// TwinCAT 3 PLC project TCP
// Title: Tc_TcpIpDevices
// Company: NewEngineer
// Author: https://github.com/phucpha
// ProjectVersion: 0.0.0.1
// Description: TC_TcpIpDevices use for Device that communicate by TCPIP.
// ProgramVersion: 3.1.4024.0
// libraries:
//   Tc2_Standard, * (Beckhoff Automation GmbH)
//   Tc2_System, * (Beckhoff Automation GmbH)
//   Tc2_TcpIp, * (Beckhoff Automation GmbH)
//   Tc3_EventLogger, * (Beckhoff Automation GmbH)
//   Tc3_Module, * (Beckhoff Automation GmbH)
//   Tc_Utilities, * (NewEngineer)
// project tree:
//   DUTs/Cognex/ E_CognexCameraGetConnectionStatus.TcDUT, E_CognexCameraGetExprStatus.TcDUT, E_CognexCameraGetFileListStatus.TcDUT, E_CognexCameraGetFileStatus.TcDUT, E_CognexCameraGetJobStatus.TcDUT, E_CognexCameraGetOnlineStatus.TcDUT, E_CognexCameraGetPositionState.TcDUT, E_CognexCameraGetPositionStatus.TcDUT, E_CognexCameraGetValueEasyBuilderStatus.TcDUT, E_CognexCameraGetValueSpreadsheetStatus.TcDUT, E_CognexCameraGetValuesState.TcDUT, E_CognexCameraGetValuesStatus.TcDUT, E_CognexCameraGetValueStatus.TcDUT, E_CognexCameraImageTriggerStatus.TcDUT, E_CognexCameraInitState.TcDUT, E_CognexCameraLoadFileStatus.TcDUT, E_CognexCameraMethodState.TcDUT, E_CognexCameraPutLiveStatus.TcDUT, E_CognexCameraPutPortnumStatus.TcDUT, E_CognexCameraPutTimeoutStatus.TcDUT, E_CognexCameraPutUpdateStatus.TcDUT, E_CognexCameraPutWatchStatus.TcDUT, E_CognexCameraResetSystemStatus.TcDUT, E_CognexCameraSetJobStatus.TcDUT, E_CognexCameraSetOnlineStatus.TcDUT, E_CognexCameraState.TcDUT, E_CognexCameraStoreFileStatus.TcDUT
//   DUTs/TcpIp/ E_TcpIpDeviceState.TcDUT, E_TcpIpDeviceStateRecive.TcDUT, E_TcpIpDeviceStateSend.TcDUT, E_TcpIpServerStateRunning.TcDUT, ST_TcpBufferData.TcDUT
//   FC/ FUN_StringToTcpBufferData.TcPOU, FUN_TcpBufferDataToString.TcPOU
//   / PlcTask.TcTTO
//   POUs/Base/Tcp Buffer/ FB_TcpBuffer.TcPOU
//   POUs/Base/Tcp Client/ FB_TcpClient.TcPOU
//   POUs/Base/Tcp Device/ FB_TcpDevice.TcPOU, I_TcpDevice.TcIO
//   POUs/Base/Tcp Server/ FB_TcpServer.TcPOU
//   POUs/Cognex/ FB_CognexCamera.TcPOU, I_CognexCamera.TcIO
//   Version/ Global_Version.TcGVL
// real-time tasks:
//   TASK PlcTask: cycle T#10ms, priority 20, ADS port 350

CONFIGURATION TCP
    RESOURCE PLC ON TwinCAT3
        TASK PlcTask(INTERVAL := T#10ms, PRIORITY := 20);
    END_RESOURCE
END_CONFIGURATION

// ---- DUTs/Cognex/E_CognexCameraGetConnectionStatus.TcDUT
{attribute 'strict'}
TYPE E_CognexCameraGetConnectionStatus :
(
	WAITING_FOR_STATUS_CODE						:= 2,
	THE_COMMAND_WAS_EXECUTED_SUCCESSFULLY		:= 1,
	UNRECOGNIZED_COMMAND 						:= 0,
	THE_CELL_ID_IS_INVALID						:= -1,
	THE_COMMAND_COULD_NOT_BE_EXECUTED 			:= -2,
	USER_DOES_NOT_HAVE_FULL_ACCESS				:= -6
);
END_TYPE

// ---- DUTs/Cognex/E_CognexCameraGetExprStatus.TcDUT
{attribute 'strict'}
TYPE E_CognexCameraGetExprStatus :
(
	WAITING_FOR_STATUS_CODE										:= 2,
	THE_COMMAND_WAS_EXECUTED_SUCCESSFULLY						:= 1,
	UNRECOGNIZED_COMMAND 										:= 0,
	THE_CELL_ID_IS_INVALID_OR_HAS_EXCEEDED_15_BYTES_IN_LENGTH	:= -1,
	THE_COMMAND_COULD_NOT_BE_EXECUTED 							:= -2
);
END_TYPE

// ---- DUTs/Cognex/E_CognexCameraGetFileListStatus.TcDUT
{attribute 'strict'}
TYPE E_CognexCameraGetFileListStatus :
(
	WAITING_FOR_STATUS_CODE									:= 2,
	THE_COMMAND_WAS_EXECUTED_SUCCESSFULLY					:= 1,
	UNRECOGNIZED_COMMAND 									:= 0,
	THE_INPUT_IS_INVALID_OR_HAS_EXCEEDED_15_BYTES_IN_LENGTH	:= -1,
	THE_ACTIVE_JOB_HAS_NOT_BEEN_SAVED 						:= -2
);
END_TYPE

// ---- DUTs/Cognex/E_CognexCameraGetFileStatus.TcDUT
{attribute 'strict'}
TYPE E_CognexCameraGetFileStatus :
(
	WAITING_FOR_STATUS_CODE						:= 2,
	THE_COMMAND_WAS_EXECUTED_SUCCESSFULLY		:= 1,
	UNRECOGNIZED_COMMAND 						:= 0,
	THE_ACTIVE_JOB_HAS_NOT_BEEN_SAVED 			:= -2
);
END_TYPE

// ---- DUTs/Cognex/E_CognexCameraGetJobStatus.TcDUT
{attribute 'strict'}
TYPE E_CognexCameraGetJobStatus :
(
	WAITING_FOR_STATUS_CODE														:= 2,
	THE_COMMAND_WAS_EXECUTED_SUCCESSFULLY										:= 1,
	UNRECOGNIZED_COMMAND 														:= 0,
	THE_ACTIVE_JOB_HAS_NOT_BEEN_SAVED_OR_DOES_NOT_HAVE_A_NUMERICAL_PREFIX		:= -2
);
END_TYPE

// ---- DUTs/Cognex/E_CognexCameraGetOnlineStatus.TcDUT
{attribute 'strict'}
TYPE E_CognexCameraGetOnlineStatus :
(
	WAITING_FOR_STATUS_CODE								:= 2,
	THE_IN_SIGHT_VISION_SYSTEM_IS_CURRENTLY_OFFLINE		:= 0,
	THE_IN_SIGHT_VISION_SYSTEM_IS_CURRENTLY_ONLINE 		:= 1
);
END_TYPE

// ---- DUTs/Cognex/E_CognexCameraGetPositionState.TcDUT
{attribute 'strict'}
TYPE E_CognexCameraGetPositionState :
(
	CAMERA_GET_POSITION_SEND_COMMAND_X				:= 0,
	CAMERA_GET_POSITION_RECEIVE_RESPONSE_X			:= 10,
	CAMERA_GET_POSITION_SEND_COMMAND_Y				:= 20,
	CAMERA_GET_POSITION_RECEIVE_RESPONSE_Y			:= 30,
	CAMERA_GET_POSITION_SEND_COMMAND_ROTATION		:= 40,
	CAMERA_GET_POSITION_RECEIVE_RESPONSE_ROTATION	:= 50,
	CAMERA_GET_POSITION_GETTING_DONE				:= 60
);
END_TYPE

// ---- DUTs/Cognex/E_CognexCameraGetPositionStatus.TcDUT
{attribute 'strict'}
TYPE E_CognexCameraGetPositionStatus :
(
	WAITING_FOR_STATUS_CODE						:= 2,
	THE_COMMAND_WAS_EXECUTED_SUCCESSFULLY		:= 1,
	UNRECOGNIZED_COMMAND 						:= 0,
	THE_SYMBOLIC_TAG_IS_INVALID					:= -1,
	THE_COMMAND_COULD_NOT_BE_EXECUTED 			:= -2,
	PRODUCT_NOT_FOUND							:= -3
);
END_TYPE

// ---- DUTs/Cognex/E_CognexCameraGetValueEasyBuilderStatus.TcDUT
{attribute 'strict'}
TYPE E_CognexCameraGetValueEasyBuilderStatus :
(
	WAITING_FOR_STATUS_CODE						:= 2,
	THE_COMMAND_WAS_EXECUTED_SUCCESSFULLY		:= 1,
	UNRECOGNIZED_COMMAND 						:= 0,
	THE_SYMBOLIC_TAG_IS_INVALID					:= -1,
	THE_COMMAND_COULD_NOT_BE_EXECUTED 			:= -2
);
END_TYPE

// ---- DUTs/Cognex/E_CognexCameraGetValueSpreadsheetStatus.TcDUT
{attribute 'strict'}
TYPE E_CognexCameraGetValueSpreadsheetStatus :
(
	WAITING_FOR_STATUS_CODE						:= 2,
	THE_COMMAND_WAS_EXECUTED_SUCCESSFULLY		:= 1,
	UNRECOGNIZED_COMMAND 						:= 0,
	THE_CELL_ID_IS_INVALID						:= -1,
	THE_COMMAND_COULD_NOT_BE_EXECUTED 			:= -2
);
END_TYPE

// ---- DUTs/Cognex/E_CognexCameraGetValuesState.TcDUT
{attribute 'strict'}
TYPE E_CognexCameraGetValuesState :
(
	CAMERA_GET_VALUES_SEND_COMMAND_VALUE_1		:= 0,
	CAMERA_GET_VALUES_RECEIVE_RESPONSE_VALUE_1	:= 10,
	CAMERA_GET_VALUES_SEND_COMMAND_VALUE_2		:= 20,
	CAMERA_GET_VALUES_RECEIVE_RESPONSE_VALUE_2	:= 30,
	CAMERA_GET_VALUES_SEND_COMMAND_VALUE_3		:= 40,
	CAMERA_GET_VALUES_RECEIVE_RESPONSE_VALUE_3	:= 50,
	CAMERA_GET_VALUES_SEND_COMMAND_VALUE_4		:= 60,
	CAMERA_GET_VALUES_RECEIVE_RESPONSE_VALUE_4	:= 70,
	CAMERA_GET_VALUES_GETTING_DONE				:= 80
);
END_TYPE

// ---- DUTs/Cognex/E_CognexCameraGetValuesStatus.TcDUT
{attribute 'strict'}
TYPE E_CognexCameraGetValuesStatus :
(
	WAITING_FOR_STATUS_CODE						:= 2,
	THE_COMMAND_WAS_EXECUTED_SUCCESSFULLY		:= 1,
	UNRECOGNIZED_COMMAND 						:= 0,
	THE_SYMBOLIC_TAG_IS_INVALID					:= -1,
	THE_COMMAND_COULD_NOT_BE_EXECUTED 			:= -2,
	ONE_OR_MORE_VALUE_IS_INVALID				:= -3
);
END_TYPE

// ---- DUTs/Cognex/E_CognexCameraGetValueStatus.TcDUT
{attribute 'strict'}
TYPE E_CognexCameraGetValueStatus :
(
	WAITING_FOR_STATUS_CODE						:= 2,
	THE_COMMAND_WAS_EXECUTED_SUCCESSFULLY		:= 1,
	UNRECOGNIZED_COMMAND 						:= 0,
	THE_CELL_ID_IS_INVALID						:= -1,
	THE_COMMAND_COULD_NOT_BE_EXECUTED 			:= -2,
	USER_DOES_NOT_HAVE_FULL_ACCESS				:= -6
);
END_TYPE

// ---- DUTs/Cognex/E_CognexCameraImageTriggerStatus.TcDUT
{attribute 'strict'}
TYPE E_CognexCameraImageTriggerStatus :
(
	WAITING_FOR_STATUS_CODE										:= 2,
	THE_COMMAND_WAS_EXECUTED_SUCCESSFULLY						:= 1,
	UNRECOGNIZED_COMMAND 										:= 0,
	THE_NUMBER_IS_EITHER_OUT_OF_RANGE_OR_NOT_AN_INTEGER 		:= -1,
	THE_COMMAND_COULD_NOT_BE_EXECUTED_OR_THE_SENSOR_IS_OFFLINE 	:= -2,
	USER_DOES_NOT_HAVE_FULL_ACCESS								:= -6
);
END_TYPE

// ---- DUTs/Cognex/E_CognexCameraInitState.TcDUT
{attribute 'strict'}
TYPE E_CognexCameraInitState :
(
	CAMERA_INIT_CONNECTION 				:= 0,
	CAMERA_INIT_CLEAR_BUFFER			:= 10,	
	CAMERA_INIT_WAIT_FOR_USERNAME 		:= 20,	
	CAMERA_INIT_WRITE_USER				:= 30,	
	CAMERA_INIT_WAIT_FOR_PASSWORD 		:= 40,	
	CAMERA_INIT_WRITE_PASSWORD			:= 50,	
	CAMERA_INIT_WAIT_FOR_CONFIRMATION	:= 60,
	CAMERA_INIT_DONE					:= 80
);
END_TYPE

// ---- DUTs/Cognex/E_CognexCameraLoadFileStatus.TcDUT
{attribute 'strict'}
TYPE E_CognexCameraLoadFileStatus :
(
	WAITING_FOR_STATUS_CODE						:= 2,
	THE_COMMAND_WAS_EXECUTED_SUCCESSFULLY		:= 1,
	UNRECOGNIZED_COMMAND 						:= 0,
	THE_FILENAME_IS_MISSING						:= -1,
	THE_JOB_FAILED_TO_LOAD 						:= -2,
	THE_VISION_SYSTEM_IS_OUT_OF_MEMORY			:= -4,
	USER_DOES_NOT_HAVE_FULL_ACCESS				:= -6
);
END_TYPE

// ---- DUTs/Cognex/E_CognexCameraMethodState.TcDUT
{attribute 'strict'}
TYPE E_CognexCameraMethodState :
(
	CAMERA_METHOD_SEND_COMMAND 			:= 0,
	CAMERA_METHOD_RECEIVE_RESPONSE 		:= 10
);
END_TYPE

// ---- DUTs/Cognex/E_CognexCameraPutLiveStatus.TcDUT
{attribute 'strict'}
TYPE E_CognexCameraPutLiveStatus :
(
	WAITING_FOR_STATUS_CODE										:= 2,
	THE_COMMAND_WAS_EXECUTED_SUCCESSFULLY						:= 1,
	UNRECOGNIZED_COMMAND 										:= 0,
	THE_INPUT_IS_INVALID_OR_HAS_EXCEEDED_15_BYTES_IN_LENGTH		:= -1,
	THE_COMMAND_COULD_NOT_BE_EXECUTED 							:= -2,
	USER_DOES_NOT_HAVE_FULL_ACCESS	 							:= -6
);
END_TYPE

// ---- DUTs/Cognex/E_CognexCameraPutPortnumStatus.TcDUT
{attribute 'strict'}
TYPE E_CognexCameraPutPortnumStatus :
(
	WAITING_FOR_STATUS_CODE										:= 2,
	THE_COMMAND_WAS_EXECUTED_SUCCESSFULLY						:= 1,
	UNRECOGNIZED_COMMAND 										:= 0,
	THE_INPUT_IS_INVALID_OR_HAS_EXCEEDED_15_BYTES_IN_LENGTH		:= -1,
	THE_COMMAND_COULD_NOT_BE_EXECUTED 							:= -2,
	USER_DOES_NOT_HAVE_FULL_ACCESS	 							:= -6
);
END_TYPE

// ---- DUTs/Cognex/E_CognexCameraPutTimeoutStatus.TcDUT
{attribute 'strict'}
TYPE E_CognexCameraPutTimeoutStatus :
(
	WAITING_FOR_STATUS_CODE										:= 2,	
	THE_COMMAND_WAS_EXECUTED_SUCCESSFULLY						:= 1,
	UNRECOGNIZED_COMMAND 										:= 0,
	THE_INPUT_IS_INVALID_OR_HAS_EXCEEDED_15_BYTES_IN_LENGTH		:= -1,
	USER_DOES_NOT_HAVE_FULL_ACCESS	 							:= -6
);
END_TYPE

// ---- DUTs/Cognex/E_CognexCameraPutUpdateStatus.TcDUT
{attribute 'strict'}
TYPE E_CognexCameraPutUpdateStatus :
(
	WAITING_FOR_STATUS_CODE										:= 2,	
	THE_COMMAND_WAS_EXECUTED_SUCCESSFULLY						:= 1,
	UNRECOGNIZED_COMMAND 										:= 0,
	THE_INPUT_IS_INVALID_OR_HAS_EXCEEDED_15_BYTES_IN_LENGTH		:= -1,
	THE_COMMAND_COULD_NOT_BE_EXECUTED 							:= -2,
	USER_DOES_NOT_HAVE_FULL_ACCESS	 							:= -6
);
END_TYPE

// ---- DUTs/Cognex/E_CognexCameraPutWatchStatus.TcDUT
{attribute 'strict'}
TYPE E_CognexCameraPutWatchStatus :
(
	WAITING_FOR_STATUS_CODE										:= 2,	
	THE_COMMAND_WAS_EXECUTED_SUCCESSFULLY						:= 1,
	UNRECOGNIZED_COMMAND 										:= 0,
	THE_INPUT_IS_INVALID_OR_HAS_EXCEEDED_15_BYTES_IN_LENGTH		:= -1,
	THE_COMMAND_COULD_NOT_BE_EXECUTED 							:= -2,
	USER_DOES_NOT_HAVE_FULL_ACCESS								:= -6
);
END_TYPE

// ---- DUTs/Cognex/E_CognexCameraResetSystemStatus.TcDUT
{attribute 'strict'}
TYPE E_CognexCameraResetSystemStatus :
(
	WAITING_FOR_STATUS_CODE					:= 2,	
	THE_COMMAND_WAS_EXECUTED_SUCCESSFULLY	:= -1,
	USER_DOES_NOT_HAVE_FULL_ACCESS			:= -6
);
END_TYPE

// ---- DUTs/Cognex/E_CognexCameraSetJobStatus.TcDUT
{attribute 'strict'}
TYPE E_CognexCameraSetJobStatus :
(
	WAITING_FOR_STATUS_CODE														:= 2,	
	THE_COMMAND_WAS_EXECUTED_SUCCESSFULLY										:= 1,
	UNRECOGNIZED_COMMAND 														:= 0,
	THE_ID_IS_LESS_THAN_0_OR_IS_NOT_AN_INTEGER									:= -1,
	THE_JOB_FAILED_TO_LOAD_THE_SENSOR_IS_ONLINE_OR_THE_FILE_WAS_NOT_FOUND		:= -2,
	THE_IN_SIGHT_SENSOR_IS_OUT_OF_MEMORY										:= -4,
	USER_DOES_NOT_HAVE_FULL_ACCESS												:= -6
);
END_TYPE

// ---- DUTs/Cognex/E_CognexCameraSetOnlineStatus.TcDUT
{attribute 'strict'}
TYPE E_CognexCameraSetOnlineStatus :
(
	WAITING_FOR_STATUS_CODE																		:= 2,	
	THE_COMMAND_WAS_EXECUTED_SUCCESSFULLY														:= 1,
	UNRECOGNIZED_COMMAND 																		:= 0,
	THE_VALUE_GIVEN_FOR_INT_IS_EITHER_OUT_OF_RANGE_OR_IS_NOT_A_VALID_INTEGER					:= -1,
	THE_COMMAND_COULD_NOT_BE_EXECUTED 															:= -2,
	THE_SENSOR_DID_NOT_GO_ONLINE_BECAUSE_IS_SET_OFFLINE_MANUAL_OR_BY_A_DISCRETE_IO_SIGNAL		:= -5,
	USER_DOES_NOT_HAVE_FULL_ACCESS																:= -6
);
END_TYPE

// ---- DUTs/Cognex/E_CognexCameraState.TcDUT
{attribute 'strict'}
TYPE E_CognexCameraState :
(
	CAMERA_UNINITIALIZED 				:= 0,	(* Not ready to work *)
	CAMERA_INITIALIZING					:= 10,	(* Preparing to work *)
	CAMERA_READY 						:= 20,	(* Ready to work *)
	CAMERA_IDLE							:= 30,	(* Waiting for commands *)
	CAMERA_RESET 						:= 40,	(* Reseting function block *)
	CAMERA_LOAD_FILE					:= 50,
	CAMERA_GET_FILE						:= 60,
	CAMERA_GET_VALUE_EASY_BUILDER		:= 70,
	CAMERA_GET_VALUE_SPREADSHEET		:= 80,
	CAMERA_SET_ONLINE					:= 90,
	CAMERA_GET_ONLINE					:= 100,
	CAMERA_RESET_SYSTEM					:= 110,
	CAMERA_GET_CONNECTIONS				:= 120,
	CAMERA_GET_EXPR						:= 130,
	CAMERA_GET_FILE_LIST				:= 140,
	CAMERA_PUT_LIVE						:= 150,
	CAMERA_PUT_PORTNUM					:= 160,
	CAMERA_PUT_TIMEOUT					:= 170,
	CAMERA_PUT_UPDATE					:= 180,
	CAMERA_PUT_WATCH					:= 190,
	CAMERA_SET_JOB						:= 200,
	CAMERA_GET_JOB						:= 210,
	CAMERA_STORE_FILE					:= 220,
	CAMERA_GET_POSITION					:= 230,
	CAMERA_IMAGE_TRIGGER				:= 240,
	CAMERA_GET_VALUES					:= 250,
	CAMERA_METHOD_DONE					:= 260,
	CAMERA_ABORTING						:= -10	(* Aborting *)
);
END_TYPE

// ---- DUTs/Cognex/E_CognexCameraStoreFileStatus.TcDUT
{attribute 'strict'}
TYPE E_CognexCameraStoreFileStatus :
(
	WAITING_FOR_STATUS_CODE																	:= 2,	
	THE_COMMAND_WAS_EXECUTED_SUCCESSFULLY													:= 1,
	UNRECOGNIZED_COMMAND 																	:= 0,
	THE_FILENAME_IS_MISSING																	:= -1,
	THE_JOB_FAILED_TO_SAVE_THE_VISION_SYSTEM_IS_ONLINE_OR_THE_FILE_WAS_NOT_FOUND 			:= -2,
	USER_DOES_NOT_HAVE_FULL_ACCESS															:= -6
);
END_TYPE

// ---- DUTs/TcpIp/E_TcpIpDeviceState.TcDUT
{attribute 'strict'}
TYPE E_TcpIpDeviceState :
(
	TCPIP_DEVICE_UNINITIALIZED 		:= 0,	(* Function block not ready to work - disconnected *)
	TCPIP_DEVICE_INITIALIZING		:= 10,	(* TCP/IP client creating client socket / TCP/IP server creating listener socket *)
	TCPIP_DEVICE_READY_INITIALIZED	:= 20,	(* Initialization finieshed successfull *)
	TCPIP_DEVICE_RUNNING			:= 30,	(* TCP/IP client data exchange with server / TCP/IP server listening for clients or data exchange with client *)
	TCPIP_DEVICE_ABORTING			:= -10	(* Closing connection and deinitialization of function block *)
);
END_TYPE

// ---- DUTs/TcpIp/E_TcpIpDeviceStateRecive.TcDUT
{attribute 'strict'}
TYPE E_TcpIpDeviceStateRecive :
(
	TCPIP_DEVICE_DATA_EXCHANGE_GET_RECIVED_DATA := 0,	(* Starting data reciving *)
	TCPIP_DEVICE_DATA_EXCHANGE_RECIVE_DONE		:= 10,	(* Waiting for any data form server *)
	TCPIP_DEVICE_DATA_EXCHANGE_WRITE_TO_BUFFER  := 20	
);
END_TYPE

// ---- DUTs/TcpIp/E_TcpIpDeviceStateSend.TcDUT
{attribute 'strict'}
TYPE E_TcpIpDeviceStateSend :
(
	TCPIP_DEVICE_DATA_EXCHANGE_GET_SEND_DATA	:= 0,	(* Append send data to clear send buffer *)
	TCPIP_DEVICE_DATA_EXCHANGE_SEND				:= 10,	(* Send data to server*)
	TCPIP_DEVICE_DATA_EXCHANGE_SEND_DONE		:= 20
);
END_TYPE

// ---- DUTs/TcpIp/E_TcpIpServerStateRunning.TcDUT
{attribute 'strict'}
TYPE E_TcpIpServerStateRunning :
(
	TCPIP_SERVER_RUNNING_START_LISTENING 		:= 0,	(* Re/Starting connection procedure *)
	TCPIP_SERVER_RUNNING_WAIT_FOR_CONNECTION	:= 10,	(* Waiting for any client *)
	TCPIP_SERVER_RUNNING_DATA_EXCHANGE 			:= 20,	(* Exchanging data with connected client *)
	TCPIP_SERVER_RUNNING_CLOSE_CONNECTION 		:= 30,	(* Closing current connection on request *)
	TCPIP_SERVER_RUNNING_CLOSE_CONNECTION_DONE	:= 40	(* Connection closed *)
);
END_TYPE

// ---- DUTs/TcpIp/ST_TcpBufferData.TcDUT
TYPE ST_TcpBufferData :
STRUCT
	arrData : ARRAY[1..8192] OF BYTE;
	iLength : UDINT;
END_STRUCT
END_TYPE

// ---- Version/Global_Version.TcGVL
{attribute 'TcGenerated'}
{attribute 'no-analysis'}
{attribute 'linkalways'}
// This function has been automatically generated from the project information.
VAR_GLOBAL CONSTANT
	{attribute 'const_non_replaced'}
	stLibVersion_Tc_TcpIpDevices : ST_LibVersion := (iMajor := 0, iMinor := 0, iBuild := 0, iRevision := 1, nFlags := 0, sVersion := '0.0.0.1');
END_VAR

// ---- POUs/Base/Tcp Device/I_TcpDevice.TcIO
INTERFACE I_TcpDevice

PROPERTY Active : REFERENCE TO BOOL
GET
END_GET
END_PROPERTY

PROPERTY AmsNetId : T_IPv4Addr
GET
END_GET
SET
END_SET
END_PROPERTY

PROPERTY Error : REFERENCE TO BOOL
GET
END_GET
END_PROPERTY

PROPERTY ErrorID : REFERENCE TO UDINT
GET
END_GET
END_PROPERTY

PROPERTY Host : T_IPv4Addr
GET
END_GET
SET
END_SET
END_PROPERTY

PROPERTY LastRecivedMessage : ST_TcpBufferData
GET
END_GET
END_PROPERTY

METHOD MR_Abort : BOOL
VAR_INPUT
END_VAR
END_METHOD

METHOD MR_FirstCycle : BOOL
VAR_INPUT
	sName 		: STRING;		(*  *)
	sHost		: T_IPv4Addr;	(*  *)
	sAmsNetID	: T_AmsNetID;	(*  *)
	iPort		: UINT;			(*  *)
	tTimeout	: TIME;			(*  *)
END_VAR
END_METHOD

METHOD MR_Init : BOOL
VAR_INPUT
END_VAR
END_METHOD

PROPERTY NextRecivedMessage : ST_TcpBufferData
GET
END_GET
END_PROPERTY

PROPERTY Port : UINT
GET
END_GET
SET
END_SET
END_PROPERTY

PROPERTY State : REFERENCE TO E_TcpIpDeviceState
GET
END_GET
END_PROPERTY

PROPERTY Timeout : TIME
GET
END_GET
SET
END_SET
END_PROPERTY

END_INTERFACE

// ---- POUs/Cognex/I_CognexCamera.TcIO
INTERFACE I_CognexCamera

PROPERTY Active : REFERENCE TO BOOL
GET
END_GET
END_PROPERTY

PROPERTY Busy : REFERENCE TO BOOL
GET
END_GET
END_PROPERTY

PROPERTY Error : REFERENCE TO BOOL
GET
END_GET
END_PROPERTY

PROPERTY ErrorID : REFERENCE TO UDINT
GET
END_GET
END_PROPERTY

METHOD MR_Abort : BOOL
VAR_INPUT
END_VAR
END_METHOD

METHOD MR_GetConnections : BOOL
END_METHOD

METHOD MR_GetExpr : BOOL
VAR_INPUT
	sCellIndexExpr	: STRING;
	iColumnExpr	: INT;
	iRowExpr	: INT;
END_VAR
END_METHOD

METHOD MR_GetFile : BOOL
END_METHOD

METHOD MR_GetFileList : BOOL
END_METHOD

METHOD MR_GetJob : BOOL
END_METHOD

METHOD MR_GetOnline : BOOL
END_METHOD

METHOD MR_GetPosition : BOOL
VAR_INPUT
	sPositionXVariable		: STRING;
	sPositionYVariable		: STRING;
	sRotationVariable		: STRING;
END_VAR

VAR_OUTPUT
	lrPositionX				: LREAL;
	lrPositionY				: LREAL;
	lrRotation				: LREAL;
END_VAR
END_METHOD

METHOD MR_GetValueEasyBuilder : BOOL
VAR_INPUT
	sEasyBuilderValueName	: STRING;
END_VAR
END_METHOD

METHOD MR_GetValues : BOOL
VAR_INPUT
	sVariable1				: STRING;
	sVariable2				: STRING;
	sVariable3				: STRING;
	sVariable4				: STRING;
END_VAR

VAR_OUTPUT
	lrValue1				: LREAL;
	lrValue2				: LREAL;
	lrValue3				: LREAL;
	lrValue4				: LREAL;	
END_VAR
END_METHOD

METHOD MR_GetValueSpreadsheet : BOOL
VAR_INPUT
	iColumnValueSpreadsheet		: INT;
	iRowValueSpreadsheet		: INT;
END_VAR
END_METHOD

METHOD MR_ImageTrigger : BOOL
END_METHOD

METHOD MR_Init : BOOL
END_METHOD

METHOD MR_LoadFile : BOOL
VAR_INPUT
	sLoadFileName	: STRING;
END_VAR
END_METHOD

METHOD MR_PutLive : BOOL
VAR_INPUT
	bEnableLiveAcquisition : INT;
END_VAR
END_METHOD

METHOD MR_PutPortnum : BOOL
VAR_INPUT
	iPortNumber : INT;
END_VAR
END_METHOD

METHOD MR_PutTimeout : BOOL
VAR_INPUT
	iTimeout 	: INT;
END_VAR
END_METHOD

METHOD MR_PutUpdate : BOOL
VAR_INPUT
	iUpdateNumber 	: INT;
END_VAR
END_METHOD

METHOD MR_PutWatch : BOOL
VAR_INPUT
	iColumnPut 		: INT;
	iRowPut 		: INT;
	iOutputEnable	: INT;
END_VAR
END_METHOD

METHOD MR_Reset : BOOL
END_METHOD

METHOD MR_ResetSystem : BOOL
END_METHOD

METHOD MR_SetJob : BOOL
VAR_INPUT
	iJobNumber 		: INT;
END_VAR
END_METHOD

METHOD MR_SetOnline : BOOL
VAR_INPUT
	bSetCameraOnline	: INT;
END_VAR
END_METHOD

METHOD MR_StoreFile : BOOL
VAR_INPUT
	sStoreFileName 	: STRING;
END_VAR
END_METHOD

PROPERTY Name : STRING
GET
END_GET
SET
END_SET
END_PROPERTY

PROPERTY ref_TcpClient : REFERENCE TO FB_TcpClient
GET
END_GET
END_PROPERTY

END_INTERFACE

// ---- FC/FUN_StringToTcpBufferData.TcPOU
(* :Description:  This function is used to convert string into bytes structure, ready to send it via TCP/IP protocole *)
FUNCTION FUN_StringToTcpBufferData : BOOL
VAR_INPUT
	sMessageAddr 	: PVOID;					(* Source string message *)
	stSendDataAddr	: PVOID;					(* Destination TCP/IP data structure *)
END_VAR
VAR
	psMessage	: POINTER TO STRING;			(* Pointer to string converted to structure *)
	pstSendData	: POINTER TO ST_TcpBufferData;	(* Pointer to structure made of string bytes *)
END_VAR

(* Check if any input address is different than zero*)
IF sMessageAddr <> 0 AND stSendDataAddr <> 0 THEN
	(* Access to adress*)
	psMessage := sMessageAddr;
	pstSendData := stSendDataAddr;
	
	pstSendData^.iLength := INT_TO_UDINT(LEN(psMessage^));
	
	(* Copy bytes from string to structure *)
	MEMCPY(destAddr := stSendDataAddr, srcAddr := sMessageAddr, n := pstSendData^.iLength);

	(* Function done *)
	FUN_StringToTcpBufferData := TRUE;
(* One of adresses was not correct *)
ELSE
	FUN_StringToTcpBufferData := FALSE;
END_IF

END_FUNCTION

// ---- FC/FUN_TcpBufferDataToString.TcPOU
(* :Description:  This function is used to convert byte structure into string text message. Structure is recived from any TCP/IP device *)
FUNCTION FUN_TcpBufferDataToString : BOOL
VAR_INPUT
	sMessageAddr		: PVOID;						(* Destination string message *)
	stReturnDataAddr	: PVOID;						(* Source TCP/IP data structure *)
END_VAR
VAR
	psMessage			: POINTER TO STRING;			(* Pointer to string converted to structure *)
	pstReturnData		: POINTER TO ST_TcpBufferData;	(* Pointer to structure made of string bytes *)
END_VAR

(* Check if any input address is different than zero*)
IF sMessageAddr <> 0 AND stReturnDataAddr <> 0 THEN
	(* Access to adress*)
	psMessage := sMessageAddr;
	pstReturnData := stReturnDataAddr;
	
	(* Clear string from any old bytes *)
	MEMSET(psMessage,0,SIZEOF(psMessage^));
	
	(* Copy bytes from string to structure *)
	MEMCPY(destAddr := psMessage, srcAddr := ADR(pstReturnData^.arrData), n:= pstReturnData^.iLength);
	
	(* Function done *)	
	FUN_TcpBufferDataToString := TRUE;
(* One of adresses was not correct *)		
ELSE
	FUN_TcpBufferDataToString := FALSE;
END_IF

END_FUNCTION

// ---- POUs/Base/Tcp Buffer/FB_TcpBuffer.TcPOU
(* 
:Description: This function block represent basic TCP/IP data buffer. It is used by all TCP devices to store data to send and recive from other devices.
*)
FUNCTION_BLOCK FB_TcpBuffer

VAR CONSTANT
	iLENGTH_OF_MESSAGE		: UDINT := 8192;
	iMAX_NUMBER_OF_MESSAGES	: UDINT := 10;
END_VAR

VAR
	arrBufferMessage	: ARRAY[0..iMAX_NUMBER_OF_MESSAGES] OF ST_TcpBufferData;
	{attribute 'hide'}
	iFirstMessageIndex	: UDINT;
	{attributee 'hide'}
	iLastMessageIndex	: UDINT;
END_VAR

(* Returns TRUE if everything went fine, FALSE if buffer is full *)
METHOD MR_Append : BOOL 
VAR_INPUT
	stData	:	ST_TcpBufferData;
END_VAR
(* Clear buffer *)
IF (arrBufferMessage[iLastMessageIndex].iLength = 0) THEN
	arrBufferMessage[iLastMessageIndex] := stData;
	MR_Append := TRUE;	
	
(* Increment one index and append data to row *)
ELSIF iLastMessageIndex < iMAX_NUMBER_OF_MESSAGES THEN
	iLastMessageIndex := iLastMessageIndex + 1;
	arrBufferMessage[iLastMessageIndex] := stData;
	MR_Append := TRUE;
	
(* Start from 0 index *)
ELSIF iFirstMessageIndex > 0 THEN
	iLastMessageIndex := 0;
	arrBufferMessage[iLastMessageIndex] := stData;
	MR_Append := TRUE;

(* Buffer is full *)	
ELSE
	MR_Append := FALSE;
	
END_IF
END_METHOD

(* Clears buffer *)
METHOD MR_Clear : BOOL
VAR_INPUT
END_VAR
MEMSET(	destAddr	:=	ADR(arrBufferMessage),
		fillByte	:=	0,
		n			:=	SIZEOF(arrBufferMessage));
		
iFirstMessageIndex := 0;
iLastMessageIndex := 0;

MR_Clear := TRUE;
END_METHOD

(* Gets last data structure from buffer *)
METHOD MR_GetLast : ST_TcpBufferData
VAR_INPUT
END_VAR
MR_GetLast := arrBufferMessage[iLastMessageIndex];
END_METHOD

(* Gets last data structure from buffer and removes it*)
METHOD MR_GetNextAndRemove : ST_TcpBufferData;
VAR_INPUT
END_VAR
(*Get data *)
MR_GetNextAndRemove := arrBufferMessage[iFirstMessageIndex];

(*Remove data from index *)
MEMSET(	destAddr	:=	ADR(arrBufferMessage[iFirstMessageIndex]), 
		fillByte	:=	0, 
		n			:=	SIZEOF(arrBufferMessage[iFirstMessageIndex]));

(* Change index of first message if it's not the only message *)
IF iFirstMessageIndex <> iLastMessageIndex THEN 
	
	(* Incerment index *)
	IF iFirstMessageIndex < iMAX_NUMBER_OF_MESSAGES THEN 
		iFirstMessageIndex := iFirstMessageIndex + 1;
	
	(* End of buffer, go to 0 *)	
	ELSE 
		iFirstMessageIndex := 0;
		
	END_IF
	
END_IF
END_METHOD

END_FUNCTION_BLOCK

// ---- POUs/Base/Tcp Client/FB_TcpClient.TcPOU
(* 
| :Description: This function block represent basic TCP/IP client. 
| Use MR_Init to connect to the server. 
| To send data to server use MR_AppendToSendBuffer, use FUN_StringToTcpBufferData to convert string into structure of bytes.
| If the lenght of LastRecivedMessage is bigger than 0 then you recived message from server, use FUN_TcpBufferDataToString to copy it to string message.
| To close the connection use MR_Abort.
*)
FUNCTION_BLOCK FB_TcpClient EXTENDS FB_TcpDevice
VAR		
	(* Function blocks *)
	fbSocketConnect : FB_SocketConnect;		(* FB used to connect the client to remote server *)
END_VAR

SUPER^();

METHOD PROTECTED MS_Aborting
IF bInitFailed THEN
	fbSocketConnect( bExecute := FALSE);
	eTcpDeviceState := TCPIP_DEVICE_UNINITIALIZED;
	
ELSE
	stSocketToClose := stHSocket;
	SUPER^.MS_Aborting();
	
END_IF
END_METHOD

(* TCP/IP client is preparing to work *)
METHOD PROTECTED MS_Initializing
SUPER^.MS_Initializing();

(* Create connection socket to remote host *)
fbSocketConnect(	sSrvNetId	:= sAmsNetID,
					sRemoteHost := sHost,
					nRemotePort := iPort,
					bExecute 	:= TRUE,
					tTimeout	:= tTimeout,
					hSocket		=> stHSocket);
						
(* Socket created *)
IF NOT fbSocketConnect.bBusy AND NOT fbSocketConnect.bError THEN
	fbSocketConnect( bExecute := FALSE);
	eTcpDeviceState := TCPIP_DEVICE_READY_INITIALIZED;
	
(*Error occured while creating client socket *)
ELSIF fbSocketConnect.bError THEN
	bError := TRUE;
	iErrorID := fbSocketConnect.nErrId;
	fbAlarmCreatingClient.ipArguments.Clear().AddUDInt(iErrorID);	
	fbAlarmCreatingClient.Raise(0);
		
END_IF
END_METHOD

END_FUNCTION_BLOCK

// ---- POUs/Base/Tcp Device/FB_TcpDevice.TcPOU
(* :Description: This function block represent basic TCP/IP device. It is used to build other function blocks like client and server. *)
FUNCTION_BLOCK ABSTRACT FB_TcpDevice IMPLEMENTS I_TcpDevice
VAR
	bFirstCycle 			: BOOL := TRUE;				(* First cycle bit *)		
	sName 					: STRING;					(* TCP/IP device name for other utilities *)
	
	(* Internal commadns *)
	bInit					: BOOL;						(* Initialize  TCP/IP device*)
	bAbort 					: BOOL;						(* Deinitialize TCP/IP device*)
	
	(* Internal status *)
	bActive					: BOOL;						(* TCP/IP device initialized and ready to work *)
	bBusy					: BOOL;						(* TCP/IP device is currently proccesing *)
	bError					: BOOL;						(* Error occured while executing *)
	bInitFailed				: BOOL;						(* Error occured while initializing *)
	iErrorID 				: UDINT;					(* Error ID*)
	eTcpDeviceState		 	: E_TcpIpDeviceState;		(* Current state of TCP/IP device*)
	eTcpDeviceSendState		: E_TcpIpDeviceStateSend;	(* Sending procedure state machine *)
	eTcpDeviceReciveState	: E_TcpIpDeviceStateRecive;	(* Reciving procedure state machine *)
	bConnectionLostError 	: BOOL;						(* Internal data exchange error - occured only in Running state *)

	(* Internal parameters *)
	sHost					: T_IPv4Addr;				(* IP address *)
	sAmsNetID 				: T_AmsNetID;				(* AMS network address *)
	iPort					: UINT;						(* Communication port *)
	tTimeout				: TIME;						(* Connection timeout *)
	stHSocket				: T_HSOCKET;				(* Socket handle *)
	stSocketToClose			: T_HSOCKET;

	(* Data buffers *)
	fbReceiveBuffer			: FB_TcpBuffer;				(* Custom buffer made to store recived data in bytes *)
	fbSendBuffer			: FB_TcpBuffer;				(* Custom buffer made to store send data in bytes *)
	
	(* Function blocks *)
	fbSocketClose 			: FB_SocketClose;			(* FB to close current connection*)
	fbSocketSend			: FB_SocketSend;			(* FB to send buffered data *)
	fbSocketRecive			: FB_SocketReceive;			(* FB to recive data*)
	
	(* Tc3 EventLogger - messages *)
	fbAlarmConnectionLost 		: FB_TcAlarm;			(*  *)
	fbAlarmClosingSocket		: FB_TcAlarm;			(*  *)
	fbAlarmCreatingListener	 	: FB_TcAlarm;			(*  *)
	fbAlarmCreatingClient		: FB_TcAlarm;			(*  *)
	fbAlarmClosingConnection	: FB_TcAlarm;			(*  *)
	fbAlarmWaitingForClient		: FB_TcAlarm;			(*  *)	

	bResetConfirmation 		: BOOL;						(*  *)
	
	rtError						: R_TRIG; 				(* Rising edge trigger for function block error *)
	
END_VAR

(* First cycle procedure *)
IF bFirstCycle THEN
	bFirstCycle := FALSE;
	
	fbAlarmConnectionLost.CreateEx( stEventEntry := TC_EVENTS.ShellTcpIpDeviceEventClass.ConnectionLost, 
									bWithConfirmation := 1,
									ipSourceInfo := 0);
									
	fbAlarmClosingSocket.CreateEx( stEventEntry := TC_EVENTS.ShellTcpIpDeviceEventClass.ClosingSocket, 
									bWithConfirmation := 1,
									ipSourceInfo := 0);			
									
	fbAlarmCreatingListener.CreateEx( stEventEntry := TC_EVENTS.ShellTcpIpDeviceEventClass.CreatingListener, 
									bWithConfirmation := 1,
									ipSourceInfo := 0);			
									
	fbAlarmCreatingClient.CreateEx( stEventEntry := TC_EVENTS.ShellTcpIpDeviceEventClass.CreatingClient, 
									bWithConfirmation := 1,
									ipSourceInfo := 0);		
									
	fbAlarmClosingConnection.CreateEx( stEventEntry := TC_EVENTS.ShellTcpIpDeviceEventClass.ClosingConnection, 
									bWithConfirmation := 1,
									ipSourceInfo := 0);		
	
	fbAlarmWaitingForClient.CreateEx( stEventEntry := TC_EVENTS.ShellTcpIpDeviceEventClass.WaitingForClient, 
									bWithConfirmation := 1,
									ipSourceInfo := 0);		
									
END_IF

(* Report errors that occur *)
rtError(CLK:=bError);

IF rtError.Q THEN 
	fbMachineLogger.MR_AddLogs(FUN_MergeStrings5(sName, ' : Error occured (error ID: ', UDINT_TO_STRING(iErrorID), ')', ''));

END_IF

(* Execute state machine *)
StateMachine();

(* Active status bit control*)
bActive := eTcpDeviceState = TCPIP_DEVICE_RUNNING OR eTcpDeviceState = TCPIP_DEVICE_ABORTING;

PROPERTY Active : REFERENCE TO BOOL
GET
Active REF= bActive;
END_GET
END_PROPERTY

PROPERTY AmsNetId : T_IPv4Addr
GET
AmsNetId := sAmsNetID;
END_GET
SET
sAmsNetID := AmsNetId;
END_SET
END_PROPERTY

PROPERTY Error : REFERENCE TO BOOL
GET
Error REF= bError;
END_GET
END_PROPERTY

PROPERTY ErrorID : REFERENCE TO UDINT
GET
ErrorID REF= iErrorID;
END_GET
END_PROPERTY

PROPERTY Host : T_IPv4Addr
GET
Host := sHost;
END_GET
SET
sHost := Host;
END_SET
END_PROPERTY

PROPERTY LastRecivedMessage : ST_TcpBufferData
GET
(*
stLastRecivedMessageTemp := fbReceiveBuffer.MR_GetLast();
LastRecivedMessage REF= stLastRecivedMessageTemp;
*)
LastRecivedMessage := fbReceiveBuffer.MR_GetLast();
END_GET
END_PROPERTY

(* Abort connection and go back to uninitialized state *)
METHOD MR_Abort : BOOL
VAR_INPUT
END_VAR
IF eTcpDeviceState > TCPIP_DEVICE_UNINITIALIZED THEN
	bAbort := TRUE;
	bInit := FALSE;
	bInitFailed := eTcpDeviceState = TCPIP_DEVICE_INITIALIZING;	
	eTcpDeviceState := TCPIP_DEVICE_ABORTING;
	fbMachineLogger.MR_AddLogs(CONCAT(sName,' : abort requested'));
	
ELSIF eTcpDeviceState = TCPIP_DEVICE_UNINITIALIZED THEN
	bAbort := FALSE;
	bInitFailed := FALSE;
	MR_Abort := TRUE;
	fbMachineLogger.MR_AddLogs(CONCAT(sName,' : abort done'));
	
END_IF
END_METHOD

(* Add data to send buffer *)
METHOD MR_AppendToSendBuffer : BOOL
VAR_INPUT
	stData : ST_TcpBufferData;
END_VAR
IF eTcpDeviceState = TCPIP_DEVICE_RUNNING THEN
	MR_AppendToSendBuffer := fbSendBuffer.MR_Append(stData);
END_IF
END_METHOD

(* Clear intearnal send and recive buffer *)
METHOD MR_ClearAllBuffers : BOOL
VAR_INPUT
END_VAR
MR_ClearAllBuffers := fbSendBuffer.MR_Clear() AND fbReceiveBuffer.MR_Clear();
END_METHOD

METHOD MR_ClearReciveBuffer : BOOL
VAR_INPUT
END_VAR
MR_ClearReciveBuffer := fbReceiveBuffer.MR_Clear();
END_METHOD

METHOD MR_ClearSendBuffer : BOOL
VAR_INPUT
END_VAR
MR_ClearSendBuffer := fbSendBuffer.MR_Clear();
END_METHOD

(* Set the initial parameters of TCP/IP device *)
METHOD MR_FirstCycle : BOOL
VAR_INPUT
	sName 		: STRING;		(* TCP/IP Device name for identyfication *)
	sHost		: T_IPv4Addr;	(* TCP/IP-Client: IP address of remote server/ TCP/IP-Server: local server IP address *)
	sAmsNetID	: T_AmsNetID;	(* TCP/IP-Client: AMS network address of remote server/ TCP/IP-Server: local server ams network address *)
	iPort		: UINT;			(* TCP/IP-Client: Port of remote server/ TCP/IP-Server: local server port *)
	tTimeout	: TIME;			(* Connection timeout *)
END_VAR
THIS^.sName 	:= sName;
THIS^.sHost 	:= sHost;
THIS^.sAmsNetID := sAmsNetID;
THIS^.iPort 	:= iPort;
THIS^.tTimeout 	:= tTimeout;
END_METHOD

(* Start initialization of TCP/IP device *)
METHOD MR_Init : BOOL
VAR_INPUT
END_VAR
IF eTcpDeviceState = TCPIP_DEVICE_UNINITIALIZED THEN
	bInit := TRUE;
	eTcpDeviceState := TCPIP_DEVICE_INITIALIZING;
	fbMachineLogger.MR_AddLogs(CONCAT(sName,' : initialization requested'));
		
ELSIF eTcpDeviceState = TCPIP_DEVICE_RUNNING THEN
	bInit := FALSE;
	MR_Init := TRUE;
	fbMachineLogger.MR_AddLogs(CONCAT(sName,' : initialization done'));	
	
END_IF
END_METHOD

(* TCP/IP device is reseting to uninitialized mode*)
METHOD PROTECTED MS_Aborting
(* Close current conncetion socket *)
fbSocketClose(	sSrvNetId 	:= sAmsNetID,
				hSocket		:= stSocketToClose,
				bExecute	:= TRUE,
				tTimeout	:= DEFAULT_ADS_TIMEOUT);
	
(* Socket closed *)				
IF NOT fbSocketClose.bBusy AND NOT fbSocketClose.bError THEN
	eTcpDeviceState := TCPIP_DEVICE_UNINITIALIZED;
	
(* Error occured while closing the socket *)
ELSIF fbSocketClose.bError THEN
	bError := TRUE;
	iErrorID := fbSocketClose.nErrId;
	fbAlarmClosingSocket.ipArguments.Clear().AddUDInt(iErrorID);	
	fbAlarmClosingSocket.Raise(0);
	
END_IF
END_METHOD

(* TCP/IP device is preparing to work *)
METHOD PROTECTED MS_Initializing
eTcpDeviceSendState := TCPIP_DEVICE_DATA_EXCHANGE_GET_SEND_DATA;
eTcpDeviceReciveState := TCPIP_DEVICE_DATA_EXCHANGE_GET_RECIVED_DATA;
END_METHOD

(* TCP/IP device is ready to work *)
METHOD PROTECTED MS_ReadyInitialized
(* Skip to device running state *)
eTcpDeviceState := TCPIP_DEVICE_RUNNING;
END_METHOD

(* TCP/IP device is working in the network *)
METHOD PROTECTED MS_Running
VAR_INST
	stDataToSend		:	ST_TcpBufferData;			(* Data to send structure *)
	stReceivedData		:	ST_TcpBufferData;			(* Recived data structure *)
	bRepeatLoop			:	BOOL;						(* Loop control bit *)
END_VAR
IF NOT bConnectionLostError THEN
	(* Send data loop *)
	REPEAT
		bRepeatLoop := FALSE;
	
		CASE eTcpDeviceSendState OF
			(*Get data to send from buffer *)
			TCPIP_DEVICE_DATA_EXCHANGE_GET_SEND_DATA:
				stDataToSend := fbSendBuffer.MR_GetNextAndRemove();
				IF stDataToSend.iLength > 0 THEN
					eTcpDeviceSendState := TCPIP_DEVICE_DATA_EXCHANGE_SEND;
					bRepeatLoop := TRUE;
					
				END_IF
			
			TCPIP_DEVICE_DATA_EXCHANGE_SEND:
				(*Send buffered data to host*)
				fbSocketSend(	sSrvNetID 	:= sAmsNetID,
								hSocket		:= stHSocket,
								cbLen		:= stDataToSend.iLength,
								pSrc		:= ADR(stDataToSend.arrData),
								bExecute	:= TRUE);
				
				eTcpDeviceSendState := TCPIP_DEVICE_DATA_EXCHANGE_SEND_DONE;
				bRepeatLoop := TRUE;
				
			TCPIP_DEVICE_DATA_EXCHANGE_SEND_DONE:	
				(* Sending done go get next data row *)			
				IF NOT fbSocketSend.bBusy AND NOT fbSocketSend.bError THEN
					fbSocketSend(bExecute := FALSE );
					eTcpDeviceSendState := TCPIP_DEVICE_DATA_EXCHANGE_GET_SEND_DATA;
					bRepeatLoop := TRUE;
						
				(* Sending in progress *)
				ELSIF fbSocketSend.bBusy AND NOT fbSocketSend.bError THEN
					eTcpDeviceSendState := TCPIP_DEVICE_DATA_EXCHANGE_SEND;
					
				(* Error occured while sending the data *)
				ELSIF fbSocketSend.bError THEN
					bError := TRUE;
					iErrorID := fbSocketSend.nErrId;
					bConnectionLostError := TRUE;
					fbAlarmConnectionLost.ipArguments.Clear().AddUDInt(iErrorID);	
					fbAlarmConnectionLost.Raise(0);
					
				END_IF
		END_CASE
	UNTIL 
		NOT bRepeatLoop
	END_REPEAT
ELSE
	fbSocketSend( bExecute := FALSE);
	
END_IF

IF NOT bConnectionLostError THEN
	(* Recive data loop *)
	REPEAT
		bRepeatLoop := FALSE;
		
		CASE eTcpDeviceReciveState OF
			TCPIP_DEVICE_DATA_EXCHANGE_GET_RECIVED_DATA:
				fbSocketRecive( 	sSrvNetId	:=	sAmsNetID,
									hSocket		:=	stHSocket,
									cbLen		:=	SIZEOF(stReceivedData.arrData),
									pDest		:=	ADR(stReceivedData.arrData),
									bExecute	:=	TRUE);
			
			eTcpDeviceReciveState := TCPIP_DEVICE_DATA_EXCHANGE_RECIVE_DONE;
			bRepeatLoop := TRUE;
			
			TCPIP_DEVICE_DATA_EXCHANGE_RECIVE_DONE:		
				IF NOT fbSocketRecive.bBusy AND NOT fbSocketRecive.bError THEN
					stReceivedData.iLength	:=	fbSocketRecive.nRecBytes;
					fbSocketRecive(	bExecute := FALSE );
					eTcpDeviceReciveState := TCPIP_DEVICE_DATA_EXCHANGE_WRITE_TO_BUFFER;
					bRepeatLoop := TRUE;
					
				ELSIF fbSocketRecive.bBusy AND NOT fbSocketRecive.bError THEN
					eTcpDeviceReciveState := TCPIP_DEVICE_DATA_EXCHANGE_GET_RECIVED_DATA;
					bRepeatLoop := FALSE;		
	
				ELSIF fbSocketRecive.bError THEN
					bError := TRUE;
					iErrorID := fbSocketRecive.nErrId;
					bConnectionLostError := TRUE;
					fbAlarmConnectionLost.ipArguments.Clear().AddUDInt(iErrorID);
					fbAlarmConnectionLost.Raise(0);
					eTcpDeviceReciveState := TCPIP_DEVICE_DATA_EXCHANGE_GET_RECIVED_DATA;
					
				END_IF
			
			TCPIP_DEVICE_DATA_EXCHANGE_WRITE_TO_BUFFER: // write data to buffer
				IF stReceivedData.iLength > 0 THEN
					fbReceiveBuffer.MR_Append(stReceivedData);
					
				END_IF
					eTcpDeviceReciveState := TCPIP_DEVICE_DATA_EXCHANGE_GET_RECIVED_DATA;
					bRepeatLoop := TRUE;
			
		END_CASE
	UNTIL 
		NOT bRepeatLoop
		
	END_REPEAT
ELSE
	fbSocketRecive(bExecute := FALSE);	
	
END_IF
END_METHOD

(* TCP/IP device is not ready to work *)
METHOD PROTECTED MS_Uninitialized
(* Reseting common function blocks *)
fbSocketSend( bExecute := FALSE);
fbSocketRecive( bExecute := FALSE);
fbSocketClose( bExecute := FALSE);

(* Clearing buffers *)
fbReceiveBuffer.MR_Clear();
fbSendBuffer.MR_Clear();

(* Reseting flags and error codes *)
bActive 				:= FALSE;
bBusy 					:= FALSE;
bError 					:= FALSE;
bInitFailed				:= FALSE;
bConnectionLostError	:= FALSE;
iErrorID 				:= 0;

(* Confirming and resetting alarms *)
fbAlarmConnectionLost.Confirm( nTimeStamp := 0);
fbAlarmClosingSocket.Confirm( nTimeStamp := 0);
fbAlarmCreatingListener.Confirm( nTimeStamp := 0);
fbAlarmCreatingClient.Confirm( nTimeStamp := 0);
fbAlarmClosingConnection.Confirm( nTimeStamp := 0);
fbAlarmWaitingForClient.Confirm( nTimeStamp := 0);

fbAlarmConnectionLost.Clear( nTimeStamp := 0, bResetConfirmation := bResetConfirmation); 
fbAlarmClosingSocket.Clear( nTimeStamp := 0, bResetConfirmation := bResetConfirmation); 
fbAlarmCreatingListener.Clear( nTimeStamp := 0, bResetConfirmation := bResetConfirmation); 
fbAlarmCreatingClient.Clear( nTimeStamp := 0, bResetConfirmation := bResetConfirmation); 
fbAlarmClosingConnection.Clear( nTimeStamp := 0, bResetConfirmation := bResetConfirmation); 
fbAlarmWaitingForClient.Clear( nTimeStamp := 0, bResetConfirmation := bResetConfirmation);
END_METHOD

PROPERTY NextRecivedMessage : ST_TcpBufferData
GET
(*
stNextRecivedMessageTemp := fbReceiveBuffer.MR_GetNextAndRemove();
NextRecivedMessage REF= stNextRecivedMessageTemp;
*)
NextRecivedMessage := fbReceiveBuffer.MR_GetNextAndRemove();
END_GET
END_PROPERTY

PROPERTY Port : UINT
GET
Port := iPort;
END_GET
SET
iPort := Port;
END_SET
END_PROPERTY

PROPERTY State : REFERENCE TO E_TcpIpDeviceState
GET
State REF= eTcpDeviceState;
END_GET
END_PROPERTY

(* Standard state machine call for TCP/IP device *)
METHOD PROTECTED StateMachine
CASE eTcpDeviceState OF
	(* TCP/IP device is not ready to work *)
	TCPIP_DEVICE_UNINITIALIZED:
		MS_Uninitialized();
	
	(* TCP/IP device is preparing to work *)	
	TCPIP_DEVICE_INITIALIZING:
		MS_Initializing();
	
	(* TCP/IP device is ready to work *)	
	TCPIP_DEVICE_READY_INITIALIZED:
		MS_ReadyInitialized();
		
	(* TCP/IP device is working in the network *)
	TCPIP_DEVICE_RUNNING:
		MS_Running();
	
	(* TCP/IP device is reseting to uninitialized mode*)	
	TCPIP_DEVICE_ABORTING:
		MS_Aborting();
		
END_CASE
END_METHOD

PROPERTY Timeout : TIME
GET
Timeout := tTimeout;
END_GET
SET
tTimeout := Timeout;
END_SET
END_PROPERTY

END_FUNCTION_BLOCK

// ---- POUs/Base/Tcp Server/FB_TcpServer.TcPOU
(* 
:Description: This function block represent basic TCP/IP client.
*)
FUNCTION_BLOCK FB_TcpServer EXTENDS FB_TcpDevice
VAR
	(* Internal command *)
	bDisconnect			: BOOL := FALSE;		(* Disconnect server from current connection *)	
	
	(* Internal parameters *)
	stHListener			: T_HSOCKET;			(* Server listener handle *)
	
	(* Internal status *)
	eTcpServerState		: E_TcpIpServerStateRunning;	(* Current server state while running *)
	
	(* Function blocks*)
	fbSocketAccept		: FB_SocketAccept;		(* FB to listen for clienncts connection requests *)
	fbSocketListen		: FB_SocketListen;		(* FB create servers listener socket *)
	
END_VAR

SUPER^();

(* Stop connection with current client and wait for another connection *)
METHOD MR_Disconnect : BOOL
VAR_INPUT
END_VAR
IF eTcpDeviceState = TCPIP_DEVICE_RUNNING AND eTcpServerState = TCPIP_SERVER_RUNNING_DATA_EXCHANGE THEN
	bDisconnect := TRUE;
	fbMachineLogger.MR_AddLogs(CONCAT(sName,' : disconnection requested'));

ELSIF eTcpDeviceState = TCPIP_DEVICE_RUNNING AND eTcpServerState = TCPIP_SERVER_RUNNING_CLOSE_CONNECTION_DONE THEN
	bDisconnect := FALSE;
	MR_Disconnect := TRUE;
	fbMachineLogger.MR_AddLogs(CONCAT(sName,' : disconnection done'));
END_IF
END_METHOD

METHOD PROTECTED MS_Aborting
IF bInitFailed THEN
	fbSocketListen( bExecute := FALSE);
	fbSocketAccept( bExecute := FALSE);
	eTcpDeviceState := TCPIP_DEVICE_UNINITIALIZED;
	
ELSE
	stSocketToClose := stHListener;
	SUPER^.MS_Aborting();
	
END_IF
END_METHOD

(* TCP/IP server is preparing to work *)
METHOD PROTECTED MS_Initializing
SUPER^.MS_Initializing();

(* Creating server listener socket at selected address and port *)
fbSocketListen( sSrvNetId	:= sAmsNetID,
				sLocalHost	:= sHost,
				nLocalPort	:= iPort,
				bExecute	:= TRUE,
				tTimeout	:= DEFAULT_ADS_TIMEOUT,
				hListener	=> stHListener);
					
(* Socket created *)	
IF NOT fbSocketListen.bBusy AND NOT fbSocketListen.bError THEN
	fbSocketListen( bExecute := FALSE);
	eTcpDeviceState := TCPIP_DEVICE_READY_INITIALIZED;
	eTcpServerState := TCPIP_SERVER_RUNNING_START_LISTENING;
		
(* Error occured while creating listener socket *)
ELSIF fbSocketListen.bError THEN	
	bError := TRUE;
	iErrorID := fbSocketListen.nErrId;
	fbAlarmCreatingListener.ipArguments.Clear().AddUDInt(iErrorID);	
	fbAlarmCreatingListener.Raise(0);
	
END_IF
END_METHOD

METHOD PROTECTED MS_Running
VAR_INST
	stDataToSend	:	ST_TcpBufferData;			(* Data to send structure *)
	stReceivedData	:	ST_TcpBufferData;			(* Recived data structure *)
	bRepeatLoop		:	BOOL;						(* Loop control bit *)
END_VAR
CASE eTcpServerState OF
	(* Reset listening FB*)
	TCPIP_SERVER_RUNNING_START_LISTENING:
		fbSocketAccept( bExecute := FALSE);
		eTcpServerState := TCPIP_SERVER_RUNNING_WAIT_FOR_CONNECTION;
	
	(* Wait for client connection *)
	TCPIP_SERVER_RUNNING_WAIT_FOR_CONNECTION:
		fbSocketAccept( sSrvNetId	:= sAmsNetID,
						hListener	:= stHListener,
						bExecute	:= TRUE,
						tTimeout	:= tTimeout);
			
		(* FB finished work without error *)			
		IF NOT fbSocketAccept.bBusy AND NOT fbSocketAccept.bError THEN
			(* Client connected *)
			IF fbSocketAccept.bAccepted THEN
				stHSocket := fbSocketAccept.hSocket;
				fbSocketAccept( bExecute := FALSE);
				
				eTcpDeviceSendState := TCPIP_DEVICE_DATA_EXCHANGE_GET_SEND_DATA;
				eTcpDeviceReciveState := TCPIP_DEVICE_DATA_EXCHANGE_GET_RECIVED_DATA;
				eTcpServerState := TCPIP_SERVER_RUNNING_DATA_EXCHANGE;
				fbMachineLogger.MR_AddLogs(CONCAT(sName,' : client connected'));
			
				(* Client not connected *)
			ELSE
				eTcpServerState := TCPIP_SERVER_RUNNING_START_LISTENING;
				
			END_IF
			
		(* Error occured while waiting for connection *)	
		ELSIF fbSocketAccept.bError THEN
			bError := TRUE;
			iErrorID := fbSocketAccept.nErrId;
			fbAlarmWaitingForClient.ipArguments.Clear().AddUDInt(iErrorID);	
			fbAlarmWaitingForClient.Raise(0);
			
		END_IF
			
	
	TCPIP_SERVER_RUNNING_DATA_EXCHANGE:
		(* Safe end of data exchange - disconnect from current connection *)
		IF bDisconnect THEN
			fbReceiveBuffer.MR_Clear();
			fbSendBuffer.MR_Clear();
			fbSocketSend(bExecute := FALSE);
			fbSocketRecive(bExecute := FALSE);
			
			IF NOT fbSocketSend.bBusy AND NOT fbSocketRecive.bBusy THEN
				eTcpServerState := TCPIP_SERVER_RUNNING_CLOSE_CONNECTION;
				
			END_IF
			
		(* Standard data exchange procedure *)
		ELSE
			SUPER^.MS_Running(); 
			
		END_IF	
	
	TCPIP_SERVER_RUNNING_CLOSE_CONNECTION:
		(* Close current connection *)
		fbSocketClose( 	sSrvNetId 	:= sAmsNetID,
						hSocket		:= stHSocket,
						bExecute	:= TRUE,
						tTimeout	:= tTimeout);
			
		(* Connection closed *)
		IF NOT fbSocketClose.bBusy AND NOT fbSocketClose.bError THEN
			fbSocketClose( bExecute := FALSE);
			eTcpServerState := TCPIP_SERVER_RUNNING_CLOSE_CONNECTION_DONE;
			
		(* Error occured while closing the connection *)
		ELSIF fbSocketClose.bError THEN
			bError := TRUE;
			iErrorID := fbSocketClose.nErrId;
			fbAlarmClosingConnection.ipArguments.Clear().AddUDInt(iErrorID);	
			fbAlarmClosingConnection.Raise(0);
			
		END_IF
	
	TCPIP_SERVER_RUNNING_CLOSE_CONNECTION_DONE:
		(* Disconnect procedure done *)
		IF NOT bDisconnect THEN
			fbSocketSend( bExecute := FALSE);
			fbSocketRecive( bExecute := FALSE);
			bError := FALSE;
			iErrorID := 0;
			bConnectionLostError := FALSE;
			eTcpServerState := TCPIP_SERVER_RUNNING_START_LISTENING;
			
		END_IF	
	
END_CASE
END_METHOD

PROPERTY ServerState : REFERENCE TO E_TcpIpServerStateRunning
GET
ServerState REF= eTcpServerState;
END_GET
END_PROPERTY

END_FUNCTION_BLOCK

// ---- POUs/Cognex/FB_CognexCamera.TcPOU
FUNCTION_BLOCK FB_CognexCamera IMPLEMENTS I_CognexCamera
VAR
	bFirstCycle 						: BOOL := TRUE;				(* First cycle bit *)		
	sName 								: STRING;					(* TCP/IP device name for other utilities *)	
 	                        			
	(* Internal status *)   			
	bActive								: BOOL;						(* TCP/IP device initialized and ready to work *)
	bBusy								: BOOL;						(* TCP/IP device is currently proccesing *)
	bError								: BOOL;						(* Error occured while executing *)
	iErrorID 							: UDINT;					(* Error ID*)
	                        			
	eCameraState		 				: E_CognexCameraState;			(* Current state of camera connection *)
	eCameraInitState					: E_CognexCameraInitState;		(* Current state of camera initialization *)
	eCameraMethodState					: E_CognexCameraMethodState;
	eCameraGetPositionState				: E_CognexCameraGetPositionState;
	eCameraGetValuesState				: E_CognexCameraGetValuesState;
	                        	
	bConnectionLostError 				: BOOL;						(* Internal data exchange error - occured only in Running state *)
	
	eCameraGetConnectionStatus			: E_CognexCameraGetConnectionStatus;
	eCameraGetExprStatus				: E_CognexCameraGetExprStatus;
	eCameraGetFileListStatus			: E_CognexCameraGetFileListStatus;
	eCameraGetFileStatus				: E_CognexCameraGetFileStatus;
	eCameraGetJobStatus 				: E_CognexCameraGetJobStatus;
	eCameraGetOnlineStatus				: E_CognexCameraGetOnlineStatus;
	eCameraGetValueEasyBuilderStatus	: E_CognexCameraGetValueEasyBuilderStatus;
	eCameraGetValueSpreadsheetStatus	: E_CognexCameraGetValueSpreadsheetStatus;
	eCameraGetValueStatus				: E_CognexCameraGetValueStatus;
	eCameraLoadFileStatus				: E_CognexCameraLoadFileStatus;
	eCameraPutLiveStatus				: E_CognexCameraPutLiveStatus;
	eCameraPutPortnumStatus				: E_CognexCameraPutPortnumStatus;
	eCameraPutTimeoutStatus				: E_CognexCameraPutTimeoutStatus;
	eCameraPutUpdateStatus				: E_CognexCameraPutUpdateStatus;
	eCameraPutWatchStatus				: E_CognexCameraPutWatchStatus;
	eCameraResetSystemStatus			: E_CognexCameraResetSystemStatus;
	eCameraSetJobStatus					: E_CognexCameraSetJobStatus;
	eCameraSetOnlineStatus				: E_CognexCameraSetOnlineStatus;
	eCameraStoreFileStatus				: E_CognexCameraStoreFileStatus;
	eCameraGetPositionStatus			: E_CognexCameraGetPositionStatus;
	eCameraImageTriggerStatus			: E_CognexCameraImageTriggerStatus;
	eCameraGetValuesStatus				: E_CognexCameraGetValuesStatus;
	
	(* Function blocks *)
	fbTcpClient 						: FB_TcpClient;				(* FB to create client connection*)
	
	(* Timers *)
	tTimeout							: TON;
	
	(* Messages buffers *)
	stSendData							: ST_TcpBufferData;		(*  *)
	stReciveData 						: ST_TcpBufferData;		(*  *)

	(* Temporary messeges *)
	sSendMessage 						: STRING;				(*  *)
	sReciveMessage						: STRING(1000);			(*  *)
	arrBufferMessage					: ARRAY[0..10] OF STRING;
	iMessageIndex	 					: INT;	
	sNewLine							: STRING := '$R$L';
	
	(* Rising edge trigger *)
	rtError								: R_TRIG; 					(* Rising edge trigger for function block error *)
	
	(* Status inormation and number *)
	iLastStatusCode						: INT; 
	sLastStatusCode						: STRING;
	                        			
	sPositionXVariable					: STRING;
	sPositionYVariable					: STRING;
	sRotationVariable					: STRING;
	                        			
	sVariable1							: STRING;
	sVariable2							: STRING;
	sVariable3							: STRING;
	sVariable4							: STRING;
	                        			
	lrPositionX							: LREAL;
	lrPositionY							: LREAL;
	lrRotation							: LREAL;
                            			
	lrValue1							: LREAL;
	lrValue2							: LREAL;
	lrValue3							: LREAL;
	lrValue4							: LREAL;
	                        			
	sPositionString						: STRING;
	sPositionStringDel					: STRING; 
	
	(* Internal variables of methods *)
	sCellIndexExpr						: STRING;
	iColumnExpr 						: INT;
	iRowExpr 							: INT;
	sEasyBuilderValueName				: STRING;
	iColumnValueSpreadsheet				: INT;
	iRowValueSpreadsheet				: INT;
	sLoadFileName						: STRING;
	bEnableLiveAcquisition				: INT;
	iPortNumber							: INT;
	iTimeout							: INT;	
	iUpdateNumber						: INT;
	iColumnPut 							: INT;
	iRowPut 							: INT;
	iOutputEnable						: INT;
	iJobNumber							: INT;
	bSetCameraOnline					: INT;
	sStoreFileName						: STRING;
END_VAR

(* First cycle procedure *)
IF bFirstCycle THEN
	bFirstCycle := FALSE;	
		
END_IF

bActive := eCameraState >= CAMERA_READY;

(* Report errors that occur *)
rtError(CLK:=bError);

IF rtError.Q THEN 
	fbMachineLogger.MR_AddLogs(FUN_MergeStrings5(sName, ' : Error occured (error ID: ', UDINT_TO_STRING(iErrorID), ')', ''));

END_IF

(* Execute TCP/IP FB and timers *)
tTimeout();
fbTcpClient();

(* Execute state machine *)
StateMachine();

PROPERTY Active : REFERENCE TO BOOL
GET
Active REF= bActive;
END_GET
END_PROPERTY

PROPERTY Busy : REFERENCE TO BOOL
GET
Busy REF= bBusy;
END_GET
END_PROPERTY

PROPERTY Error : REFERENCE TO BOOL
GET
Error REF= bError;
END_GET
END_PROPERTY

PROPERTY ErrorID : REFERENCE TO UDINT
GET
ErrorID REF= iErrorID;
END_GET
END_PROPERTY

METHOD M_ResetParameters : BOOL
VAR_INPUT
END_VAR
eCameraGetConnectionStatus			:= 2;
eCameraGetExprStatus				:= 2;
eCameraGetFileListStatus			:= 2;
eCameraGetFileStatus				:= 2;
eCameraGetJobStatus 				:= 2;
eCameraGetOnlineStatus				:= 2;
eCameraGetValueEasyBuilderStatus	:= 2;
eCameraGetValueSpreadsheetStatus	:= 2;
eCameraGetValueStatus				:= 2;
eCameraLoadFileStatus				:= 2;
eCameraPutLiveStatus				:= 2;
eCameraPutPortnumStatus				:= 2;
eCameraPutTimeoutStatus				:= 2;
eCameraPutUpdateStatus				:= 2;
eCameraPutWatchStatus				:= 2;
eCameraResetSystemStatus			:= 2;
eCameraSetJobStatus					:= 2;
eCameraSetOnlineStatus				:= 2;
eCameraStoreFileStatus				:= 2;
eCameraGetPositionStatus			:= 2;
eCameraImageTriggerStatus			:= 2;
eCameraGetValuesStatus				:= 2;

sSendMessage 						:= '';
sReciveMessage						:= '';
iMessageIndex	 					:= 0;	

(* Status inormation and number *)
iLastStatusCode						:= 0; 
sLastStatusCode						:= '';
	
(* Internal variables of methods *)
sCellIndexExpr						:= '';
iColumnExpr 						:= 0;
iRowExpr 							:= 0;
sEasyBuilderValueName				:= '';
iColumnValueSpreadsheet				:= 0;
iRowValueSpreadsheet				:= 0;
sLoadFileName						:= '';
bEnableLiveAcquisition				:= 0;
iPortNumber							:= 0;
iTimeout							:= 0;	
iUpdateNumber						:= 0;
iColumnPut 							:= 0;
iRowPut 							:= 0;
iOutputEnable						:= 0;
iJobNumber							:= 0;
bSetCameraOnline					:= 0;
sStoreFileName						:= '';
	
sPositionXVariable					:= '';
sPositionYVariable					:= '';
sRotationVariable					:= '';

sVariable1							:= '';
sVariable2							:= '';
sVariable3							:= '';
sVariable4							:= '';

lrPositionX							:= 0.0;
lrPositionY							:= 0.0;
lrRotation							:= 0.0;

lrValue1							:= 0.0;
lrValue2							:= 0.0;			
lrValue3							:= 0.0;
lrValue4							:= 0.0;

sPositionString						:= '';
sPositionStringDel					:= '';	

(* Internal status *)
bActive								:= 0;						(* TCP/IP device initialized and ready to work *)
bBusy								:= 0;						(* TCP/IP device is currently proccesing *)
bError								:= 0;						(* Error occured while executing *)
iErrorID 							:= 0;					(* Error ID*)

	
eCameraGetPositionState := 0;
eCameraGetValuesState := 0;
eCameraMethodState := 0;
eCameraInitState := 0;

M_ResetParameters := TRUE;
END_METHOD

METHOD MR_Abort : BOOL
VAR_INPUT
END_VAR
IF eCameraState >= CAMERA_READY THEN
	bBusy := TRUE;
	MR_Abort := FALSE;
	eCameraState := CAMERA_ABORTING;
	fbMachineLogger.MR_AddLogs(CONCAT(sName,' : abort requested'));	
	
ELSIF eCameraState = CAMERA_UNINITIALIZED THEN
	bBusy := FALSE;
	MR_Abort := TRUE;
	fbMachineLogger.MR_AddLogs(CONCAT(sName,' : abort done'));	
	
END_IF
END_METHOD

METHOD MR_FirstCycle : BOOL
VAR_INPUT
	sCameraName 	: STRING;		(*  *)
	sClientHost		: T_IPv4Addr;	(*  *)
	sClientAmsNetID : T_AmsNetID;	(*  *)
	iClientPort		: UINT;			(*  *)
	tTimeout		: TIME;			(*  *)
END_VAR
(* Set fixture name *)
THIS^.sName := sCameraName;

(* Set fixture server initial parameters *)
THIS^.fbTcpClient.MR_FirstCycle(	sName 		:= CONCAT('TCP/IP client of ',sCameraName),
									sHost		:= sClientHost,
									sAmsNetID	:= sClientAmsNetID,
									iPort 		:= iClientPort,
									tTimeout 	:= tTimeout);
END_METHOD

METHOD MR_GetConnections : BOOL
IF eCameraState = CAMERA_IDLE THEN
	bBusy := TRUE;
	MR_GetConnections := FALSE;
	eCameraState := CAMERA_GET_CONNECTIONS;
	fbMachineLogger.MR_AddLogs(CONCAT(sName,' : returning current connection information requested'));	
	
ELSIF eCameraState = CAMERA_METHOD_DONE THEN
	bBusy := FALSE;
	MR_GetConnections := TRUE;
	fbMachineLogger.MR_AddLogs(CONCAT(sName,' : returning current connection information done'));	
	
END_IF
END_METHOD

METHOD MR_GetExpr : BOOL
VAR_INPUT
	sCellIndexExpr	: STRING;
	iColumnExpr	: INT;
	iRowExpr	: INT;
END_VAR
IF eCameraState = CAMERA_IDLE THEN
	THIS^.sCellIndexExpr := sCellIndexExpr;
	THIS^.iColumnExpr	:= iColumnExpr;
	THIS^.iRowExpr	:= iRowExpr;	
	bBusy := TRUE;
	MR_GetExpr := FALSE;
	eCameraState := CAMERA_GET_EXPR;
	fbMachineLogger.MR_AddLogs(CONCAT(sName,' : returning the parameters or value stored in the cell requested'));	
	
ELSIF eCameraState = CAMERA_METHOD_DONE THEN
	bBusy := FALSE;
	MR_GetExpr := TRUE;
	fbMachineLogger.MR_AddLogs(CONCAT(sName,' : returning the parameters or value stored in the cell done'));	
	
END_IF
END_METHOD

METHOD MR_GetFile : BOOL
IF eCameraState = CAMERA_IDLE THEN
	bBusy := TRUE;
	MR_GetFile := FALSE;
	eCameraState := CAMERA_GET_FILE;
	fbMachineLogger.MR_AddLogs(CONCAT(sName,' : getting the filename of the active job requested'));	
	
ELSIF eCameraState = CAMERA_METHOD_DONE THEN
	bBusy := FALSE;
	MR_GetFile := TRUE;
	fbMachineLogger.MR_AddLogs(CONCAT(sName,' : getting the filename of the active job done'));	
	
END_IF
END_METHOD

METHOD MR_GetFileList : BOOL
IF eCameraState = CAMERA_IDLE THEN
	bBusy := TRUE;
	MR_GetFileList := FALSE;
	eCameraState := CAMERA_GET_FILE_LIST;
	fbMachineLogger.MR_AddLogs(CONCAT(sName,' : returning the number and names of files stored in memory requested'));	
	
ELSIF eCameraState = CAMERA_METHOD_DONE THEN
	bBusy := FALSE;
	MR_GetFileList := TRUE;
	fbMachineLogger.MR_AddLogs(CONCAT(sName,' : returning the number and names of files stored in memory done'));	
	
END_IF
END_METHOD

METHOD MR_GetJob : BOOL
IF eCameraState = CAMERA_IDLE THEN
	bBusy := TRUE;
	MR_GetJob := FALSE;
	eCameraState := CAMERA_GET_JOB;
	fbMachineLogger.MR_AddLogs(CONCAT(sName,' : returning a status code (ID) of the active job requested'));	
	
ELSIF eCameraState = CAMERA_METHOD_DONE THEN
	bBusy := FALSE;
	MR_GetJob := TRUE;
	fbMachineLogger.MR_AddLogs(CONCAT(sName,' : returning a status code (ID) of the active job done'));	
	
END_IF
END_METHOD

METHOD MR_GetOnline : BOOL
IF eCameraState = CAMERA_IDLE THEN
	bBusy := TRUE;
	MR_GetOnline := FALSE;
	eCameraState := CAMERA_GET_ONLINE;
	fbMachineLogger.MR_AddLogs(CONCAT(sName,' : returning the online state of the vision system requested'));	
	
ELSIF eCameraState = CAMERA_METHOD_DONE THEN
	bBusy := FALSE;
	MR_GetOnline := TRUE;
	fbMachineLogger.MR_AddLogs(CONCAT(sName,' :  returning the online state of the vision system done'));	
	
END_IF
END_METHOD

METHOD MR_GetPosition : BOOL
VAR_INPUT
	sPositionXVariable		: STRING;
	sPositionYVariable		: STRING;
	sRotationVariable		: STRING;
END_VAR

VAR_OUTPUT
	lrPositionX				: LREAL;
	lrPositionY				: LREAL;
	lrRotation				: LREAL;
END_VAR
IF eCameraState = CAMERA_IDLE THEN
	THIS^.sPositionXVariable := sPositionXVariable;
	THIS^.sPositionYVariable := sPositionYVariable;
	THIS^.sRotationVariable := sRotationVariable;
	bBusy := TRUE;
	MR_GetPosition := FALSE;
	eCameraState := CAMERA_GET_POSITION;
	fbMachineLogger.MR_AddLogs(CONCAT(sName,' : getting current position of the product requested'));	
	
ELSIF eCameraState = CAMERA_METHOD_DONE THEN
	lrPositionX := THIS^.lrPositionX;
	lrPositionY := THIS^.lrPositionY;
	lrRotation := THIS^.lrRotation;
	bBusy := FALSE;
	MR_GetPosition := TRUE;
	fbMachineLogger.MR_AddLogs(CONCAT(sName,' : getting current position of the product done'));	
	
END_IF
END_METHOD

METHOD MR_GetValueEasyBuilder : BOOL
VAR_INPUT
	sEasyBuilderValueName	: STRING;
END_VAR
IF eCameraState = CAMERA_IDLE THEN
	THIS^.sEasyBuilderValueName := sEasyBuilderValueName;
	bBusy := TRUE;
	MR_GetValueEasyBuilder := FALSE;
	eCameraState := CAMERA_GET_VALUE_EASY_BUILDER;
	fbMachineLogger.MR_AddLogs(CONCAT(sName,' : returning the tool result or job data in EasyBuilder requested'));	
	
ELSIF eCameraState = CAMERA_METHOD_DONE THEN
	bBusy := FALSE;
	MR_GetValueEasyBuilder := TRUE;
	fbMachineLogger.MR_AddLogs(CONCAT(sName,' : returning the tool result or job data in EasyBuilder done'));	
	
END_IF
END_METHOD

METHOD MR_GetValues : BOOL
VAR_INPUT
	sVariable1				: STRING;
	sVariable2				: STRING;
	sVariable3				: STRING;
	sVariable4				: STRING;
END_VAR

VAR_OUTPUT
	lrValue1				: LREAL;
	lrValue2				: LREAL;
	lrValue3				: LREAL;
	lrValue4				: LREAL;	
END_VAR
IF eCameraState = CAMERA_IDLE THEN
	THIS^.sVariable1 := sVariable1;
	THIS^.sVariable2 := sVariable2;
	THIS^.sVariable3 := sVariable3;
	THIS^.sVariable4 := sVariable4;
	bBusy := TRUE;
	MR_GetValues := FALSE;
	eCameraState := CAMERA_GET_VALUES;
	fbMachineLogger.MR_AddLogs(CONCAT(sName,' : getting values from camera requested'));	
	
ELSIF eCameraState = CAMERA_METHOD_DONE THEN
	lrValue1 := THIS^.lrValue1;
	lrValue2 := THIS^.lrValue2;
	lrValue3 := THIS^.lrValue3;
	lrValue4 := THIS^.lrValue4;
	bBusy := FALSE;
	MR_GetValues := TRUE;
	fbMachineLogger.MR_AddLogs(CONCAT(sName,' : getting values from camera done'));	
	
END_IF
END_METHOD

METHOD MR_GetValueSpreadsheet : BOOL
VAR_INPUT
	iColumnValueSpreadsheet		: INT;
	iRowValueSpreadsheet		: INT;
END_VAR
IF eCameraState = CAMERA_IDLE THEN
	THIS^.iColumnValueSpreadsheet := iColumnValueSpreadsheet;
	THIS^.iRowValueSpreadsheet := iRowValueSpreadsheet;
	bBusy := TRUE;
	MR_GetValueSpreadsheet := FALSE;
	eCameraState := CAMERA_GET_VALUE_SPREADSHEET;
	fbMachineLogger.MR_AddLogs(CONCAT(sName,' : returning the tool result or job data in the Spreadsheet requested'));	
	
ELSIF eCameraState = CAMERA_METHOD_DONE THEN
	bBusy := FALSE;
	MR_GetValueSpreadsheet := TRUE;
	fbMachineLogger.MR_AddLogs(CONCAT(sName,' : returning the tool result or job data in the Spreadsheet done'));	
	
END_IF
END_METHOD

METHOD MR_ImageTrigger : BOOL
IF eCameraState = CAMERA_IDLE THEN
	bBusy := TRUE;
	MR_ImageTrigger := FALSE;
	eCameraState := CAMERA_IMAGE_TRIGGER;
	fbMachineLogger.MR_AddLogs(CONCAT(sName,' : image trigger requested'));	
	
ELSIF eCameraState = CAMERA_METHOD_DONE THEN
	bBusy := FALSE;
	MR_ImageTrigger := TRUE;
	fbMachineLogger.MR_AddLogs(CONCAT(sName,' : image trigger done'));	
	
END_IF
END_METHOD

METHOD MR_Init : BOOL
IF eCameraState = CAMERA_UNINITIALIZED THEN
	bBusy := TRUE;
	MR_Init := FALSE;
	eCameraState := CAMERA_INITIALIZING;
	fbMachineLogger.MR_AddLogs(CONCAT(sName,' : initializing requested'));	
	
ELSIF eCameraState >= CAMERA_READY THEN
	bBusy := FALSE;
	MR_Init := TRUE;
	fbMachineLogger.MR_AddLogs(CONCAT(sName,' : initializing done'));	
	
END_IF
END_METHOD

METHOD MR_LoadFile : BOOL
VAR_INPUT
	sLoadFileName	: STRING;
END_VAR
IF eCameraState = CAMERA_IDLE THEN
	THIS^.sLoadFileName := sLoadFileName;
	bBusy := TRUE;
	MR_LoadFile := FALSE;
	eCameraState := CAMERA_LOAD_FILE;
	fbMachineLogger.MR_AddLogs(CONCAT(sName,' : loading the specified job from flash memory requested'));	

ELSIF eCameraState = CAMERA_METHOD_DONE THEN
	bBusy := FALSE;
	MR_LoadFile := TRUE;
	fbMachineLogger.MR_AddLogs(CONCAT(sName,' :  loading the specified job from flash memory done'));	
	
END_IF
END_METHOD

METHOD MR_PutLive : BOOL
VAR_INPUT
	bEnableLiveAcquisition : INT;
END_VAR
IF eCameraState = CAMERA_IDLE THEN
	THIS^.bEnableLiveAcquisition := bEnableLiveAcquisition;
	bBusy := TRUE;
	MR_PutLive := FALSE;
	eCameraState := CAMERA_PUT_LIVE;
	fbMachineLogger.MR_AddLogs(CONCAT(sName,' : turning live acquisition mode on or off requested'));	
	
ELSIF eCameraState = CAMERA_METHOD_DONE THEN
	bBusy := FALSE;
	MR_PutLive := TRUE;
	fbMachineLogger.MR_AddLogs(CONCAT(sName,' : turning live acquisition mode on or off done'));	
	
END_IF
END_METHOD

METHOD MR_PutPortnum : BOOL
VAR_INPUT
	iPortNumber : INT;
END_VAR
IF eCameraState = CAMERA_IDLE THEN
	THIS^.iPortNumber := iPortNumber;
	bBusy := TRUE;
	MR_PutPortnum := FALSE;
	eCameraState := CAMERA_PUT_PORTNUM;
	fbMachineLogger.MR_AddLogs(CONCAT(sName,' : specifying the communication port number requested'));	
	
ELSIF eCameraState = CAMERA_METHOD_DONE THEN
	bBusy := FALSE;
	MR_PutPortnum := TRUE;
	fbMachineLogger.MR_AddLogs(CONCAT(sName,' : specifying the communication port number done'));	
	
END_IF
END_METHOD

METHOD MR_PutTimeout : BOOL
VAR_INPUT
	iTimeout 	: INT;
END_VAR
IF eCameraState = CAMERA_IDLE THEN
	THIS^.iTimeout := iTimeout;
	bBusy := TRUE;
	MR_PutTimeout := FALSE;
	eCameraState := CAMERA_PUT_TIMEOUT;
	fbMachineLogger.MR_AddLogs(CONCAT(sName,' : specifying a port connection timeout requested'));	
	
ELSIF eCameraState = CAMERA_METHOD_DONE THEN
	bBusy := FALSE;
	MR_PutTimeout := TRUE;
	fbMachineLogger.MR_AddLogs(CONCAT(sName,' : specifying a port connection timeout done'));	
	
END_IF
END_METHOD

METHOD MR_PutUpdate : BOOL
VAR_INPUT
	iUpdateNumber 	: INT;
END_VAR
IF eCameraState = CAMERA_IDLE THEN
	THIS^.iUpdateNumber := iUpdateNumber;
	bBusy := TRUE;
	MR_PutUpdate := FALSE;
	eCameraState := CAMERA_PUT_UPDATE;
	fbMachineLogger.MR_AddLogs(CONCAT(sName,' : updating the GUI requested'));	
	
ELSIF eCameraState = CAMERA_METHOD_DONE THEN
	bBusy := FALSE;
	MR_PutUpdate := TRUE;
	fbMachineLogger.MR_AddLogs(CONCAT(sName,' : updating the GUI done'));	
	
END_IF
END_METHOD

METHOD MR_PutWatch : BOOL
VAR_INPUT
	iColumnPut 		: INT;
	iRowPut 		: INT;
	iOutputEnable	: INT;
END_VAR
IF eCameraState = CAMERA_IDLE THEN
	THIS^.iColumnPut := iColumnPut;
	THIS^.iRowPut := iRowPut;
	THIS^.iOutputEnable := iOutputEnable;
	bBusy := TRUE;
	MR_PutWatch := FALSE;
	eCameraState := CAMERA_PUT_WATCH;
	fbMachineLogger.MR_AddLogs(CONCAT(sName,' : returning the value contained in the specified cell each time the cell is updated requested'));	
	
ELSIF eCameraState = CAMERA_METHOD_DONE THEN
	bBusy := FALSE;
	MR_PutWatch := TRUE;
	fbMachineLogger.MR_AddLogs(CONCAT(sName,' : returning the value contained in the specified cell each time the cell is updated done'));	
	
END_IF
END_METHOD

METHOD MR_Reset : BOOL
IF eCameraState >= CAMERA_READY AND eCameraState <> CAMERA_METHOD_DONE THEN
	bBusy := TRUE;
	MR_Reset := FALSE;
	eCameraState := CAMERA_RESET;	
	fbMachineLogger.MR_AddLogs(CONCAT(sName,' : camera FB reset requested'));	
	
ELSIF eCameraState = CAMERA_METHOD_DONE THEN
	bBusy := FALSE;
	MR_Reset := TRUE;
	fbMachineLogger.MR_AddLogs(CONCAT(sName,' : camera FB reset done'));	
	
END_IF
END_METHOD

METHOD MR_ResetSystem : BOOL
IF eCameraState = CAMERA_IDLE THEN
	bBusy := TRUE;
	MR_ResetSystem := FALSE;
	eCameraState := CAMERA_RESET_SYSTEM;
	fbMachineLogger.MR_AddLogs(CONCAT(sName,' : resetting the In-Sight sensor requested'));	
	
ELSIF eCameraState = CAMERA_METHOD_DONE THEN
	bBusy := FALSE;
	MR_ResetSystem := TRUE;
	fbMachineLogger.MR_AddLogs(CONCAT(sName,' : resetting the In-Sight sensor done'));	
	
END_IF
END_METHOD

METHOD MR_SetJob : BOOL
VAR_INPUT
	iJobNumber 		: INT;
END_VAR
IF eCameraState = CAMERA_IDLE THEN
	THIS^.iJobNumber := iJobNumber;
	bBusy := TRUE;
	MR_SetJob := FALSE;
	eCameraState := CAMERA_SET_JOB;
	fbMachineLogger.MR_AddLogs(CONCAT(sName,' : loading a job from one of the job slots in flash memory on the In-Sight sensor requested'));	
	
ELSIF eCameraState = CAMERA_METHOD_DONE THEN
	bBusy := FALSE;
	MR_SetJob := TRUE;
	fbMachineLogger.MR_AddLogs(CONCAT(sName,' : loading a job from one of the job slots in flash memory on the In-Sight sensor done'));	
	
END_IF
END_METHOD

METHOD MR_SetOnline : BOOL
VAR_INPUT
	bSetCameraOnline	: INT;
END_VAR
IF eCameraState = CAMERA_IDLE THEN
	THIS^.bSetCameraOnline := bSetCameraOnline;
	bBusy := TRUE;
	MR_SetOnline := FALSE;
	eCameraState := CAMERA_SET_ONLINE;
	fbMachineLogger.MR_AddLogs(CONCAT(sName,' : setting the In-Sight sensor into Online or Offline mode requested'));	
	
ELSIF eCameraState = CAMERA_METHOD_DONE THEN
	bBusy := FALSE;
	MR_SetOnline := TRUE;
	fbMachineLogger.MR_AddLogs(CONCAT(sName,' : setting the In-Sight sensor into Online or Offline mode done'));	
	
END_IF
END_METHOD

METHOD MR_StoreFile : BOOL
VAR_INPUT
	sStoreFileName 	: STRING;
END_VAR
IF eCameraState = CAMERA_IDLE THEN
	THIS^.sStoreFileName := sStoreFileName;
	bBusy := TRUE;
	MR_StoreFile := FALSE;
	eCameraState := CAMERA_STORE_FILE;
	fbMachineLogger.MR_AddLogs(CONCAT(sName,' : saving the current job in flash memory on the In-Sight vision system requested'));	
	
ELSIF eCameraState = CAMERA_METHOD_DONE THEN
	bBusy := FALSE;
	MR_StoreFile := TRUE;
	fbMachineLogger.MR_AddLogs(CONCAT(sName,' : saving the current job in flash memory on the In-Sight vision system done'));	
	
END_IF
END_METHOD

METHOD PROTECTED MS_Aborting
fbTcpClient.MR_Abort();

IF NOT fbTcpClient.Active THEN 
	IF M_ResetParameters() THEN
		eCameraState := CAMERA_UNINITIALIZED;
		
	END_IF	
END_IF
END_METHOD

METHOD PROTECTED MS_GetConnections
CASE eCameraMethodState OF
	CAMERA_METHOD_SEND_COMMAND:
		MEMSET(ADR(sSendMessage),0,SIZEOF(sSendMessage));
		sSendMessage := 'Get Connections$R$L';
		FUN_StringToTcpBufferData(ADR(sSendMessage),ADR(stSendData));
		
		IF fbTcpClient.MR_AppendToSendBuffer(stSendData) THEN
			eCameraMethodState := CAMERA_METHOD_RECEIVE_RESPONSE;
							
		END_IF

	CAMERA_METHOD_RECEIVE_RESPONSE:
		stReciveData := fbTcpClient.NextRecivedMessage;
		
		IF stReciveData.iLength > 0 THEN
			MEMSET(ADR(sReciveMessage),0,SIZEOF(sReciveMessage));
			FUN_TcpBufferDataToString(ADR(sReciveMessage),ADR(stReciveData));
			MEMCPY(ADR(sLastStatusCode),ADR(sReciveMessage),2);
			iLastStatusCode := STRING_TO_INT(sLastStatusCode);
			
			IF iLastStatusCode = 1 THEN 
				eCameraGetConnectionStatus := 1;
				
			ELSIF iLastStatusCode = 0 THEN
				eCameraGetConnectionStatus := 0;
				
			ELSIF iLastStatusCode = -1 THEN
				eCameraGetConnectionStatus := -1;
				
			ELSIF iLastStatusCode = -2 THEN
				eCameraGetConnectionStatus := -2;
				
			ELSIF iLastStatusCode = -6 THEN
				eCameraGetConnectionStatus := -6;
				
			END_IF	
			eCameraMethodState := CAMERA_METHOD_SEND_COMMAND;
			eCameraState := CAMERA_METHOD_DONE;

		END_IF
END_CASE
END_METHOD

METHOD PROTECTED MS_GetExpr
CASE eCameraMethodState OF
	CAMERA_METHOD_SEND_COMMAND:
		MEMSET(ADR(sSendMessage),0,SIZEOF(sSendMessage));
		sSendMessage := FUN_MergeStrings5('Get Expr ',sCellIndexExpr ,CONCAT(TO_STRING(iColumnExpr), TO_STRING(iRowExpr)), '$R$L', '');
		FUN_StringToTcpBufferData(ADR(sSendMessage),ADR(stSendData));
		
		IF fbTcpClient.MR_AppendToSendBuffer(stSendData) THEN
			eCameraMethodState := CAMERA_METHOD_RECEIVE_RESPONSE;
							
		END_IF

	CAMERA_METHOD_RECEIVE_RESPONSE:
		stReciveData := fbTcpClient.NextRecivedMessage;
		
		IF stReciveData.iLength > 0 THEN
			MEMSET(ADR(sReciveMessage),0,SIZEOF(sReciveMessage));
			FUN_TcpBufferDataToString(ADR(sReciveMessage),ADR(stReciveData));
			MEMCPY(ADR(sLastStatusCode),ADR(sReciveMessage),2);
			iLastStatusCode := STRING_TO_INT(sLastStatusCode);
			
			IF iLastStatusCode = 1 THEN 
				eCameraGetExprStatus := 1;
				
			ELSIF iLastStatusCode = 0 THEN
				eCameraGetExprStatus := 0;
				
			ELSIF iLastStatusCode = -1 THEN
				eCameraGetExprStatus := -1;
				
			ELSIF iLastStatusCode = -2 THEN
				eCameraGetExprStatus := -2;
				
			END_IF	
			eCameraMethodState := CAMERA_METHOD_SEND_COMMAND;
			eCameraState := CAMERA_METHOD_DONE;

		END_IF
END_CASE
END_METHOD

METHOD PROTECTED MS_GetFile
CASE eCameraMethodState OF
	CAMERA_METHOD_SEND_COMMAND:
		MEMSET(ADR(sSendMessage),0,SIZEOF(sSendMessage));
		sSendMessage := 'GF$R$L';
		FUN_StringToTcpBufferData(ADR(sSendMessage),ADR(stSendData));
		
		IF fbTcpClient.MR_AppendToSendBuffer(stSendData) THEN
			eCameraMethodState := CAMERA_METHOD_RECEIVE_RESPONSE;
							
		END_IF

	CAMERA_METHOD_RECEIVE_RESPONSE:
		stReciveData := fbTcpClient.NextRecivedMessage;
		
		IF stReciveData.iLength > 0 THEN
			MEMSET(ADR(sReciveMessage),0,SIZEOF(sReciveMessage));
			FUN_TcpBufferDataToString(ADR(sReciveMessage),ADR(stReciveData));
			MEMCPY(ADR(sLastStatusCode),ADR(sReciveMessage),2);
			iLastStatusCode := STRING_TO_INT(sLastStatusCode);
			
			IF iLastStatusCode = 1 THEN 
				eCameraGetFileStatus := 1;
				
			ELSIF iLastStatusCode = 0 THEN
				eCameraGetFileStatus := 0;
				
			ELSIF iLastStatusCode = -2 THEN
				eCameraGetFileStatus := -2;
				
			END_IF	
			eCameraMethodState := CAMERA_METHOD_SEND_COMMAND;
			eCameraState := CAMERA_METHOD_DONE;

		END_IF
END_CASE
END_METHOD

METHOD PROTECTED MS_GetFileList
CASE eCameraMethodState OF
	CAMERA_METHOD_SEND_COMMAND:
		MEMSET(ADR(sSendMessage),0,SIZEOF(sSendMessage));
		sSendMessage := 'Get Filelist$R$L';
		FUN_StringToTcpBufferData(ADR(sSendMessage),ADR(stSendData));
		
		IF fbTcpClient.MR_AppendToSendBuffer(stSendData) THEN
			eCameraMethodState := CAMERA_METHOD_RECEIVE_RESPONSE;
							
		END_IF

	CAMERA_METHOD_RECEIVE_RESPONSE:
		stReciveData := fbTcpClient.NextRecivedMessage;
		
		IF stReciveData.iLength > 0 THEN
			MEMSET(ADR(sReciveMessage),0,SIZEOF(sReciveMessage));
			FUN_TcpBufferDataToString(ADR(sReciveMessage),ADR(stReciveData));
			MEMCPY(ADR(sLastStatusCode),ADR(sReciveMessage),2);
			iLastStatusCode := STRING_TO_INT(sLastStatusCode);
			
			IF iLastStatusCode = 1 THEN 
				eCameraGetFileListStatus := 1;
				
			ELSIF iLastStatusCode = 0 THEN
				eCameraGetFileListStatus := 0;
				
			ELSIF iLastStatusCode = -1 THEN
				eCameraGetFileListStatus := -1;
				
			ELSIF iLastStatusCode = -2 THEN
				eCameraGetFileListStatus := -2;
				
			END_IF	
			eCameraMethodState := CAMERA_METHOD_SEND_COMMAND;
			eCameraState := CAMERA_METHOD_DONE;

		END_IF
END_CASE
END_METHOD

METHOD PROTECTED MS_GetJob
CASE eCameraMethodState OF
	CAMERA_METHOD_SEND_COMMAND:
		MEMSET(ADR(sSendMessage),0,SIZEOF(sSendMessage));
		sSendMessage := 'GJ$R$L';
		FUN_StringToTcpBufferData(ADR(sSendMessage),ADR(stSendData));
		
		IF fbTcpClient.MR_AppendToSendBuffer(stSendData) THEN
			eCameraMethodState := CAMERA_METHOD_RECEIVE_RESPONSE;
							
		END_IF

	CAMERA_METHOD_RECEIVE_RESPONSE:
		stReciveData := fbTcpClient.NextRecivedMessage;
		
		IF stReciveData.iLength > 0 THEN
			MEMSET(ADR(sReciveMessage),0,SIZEOF(sReciveMessage));
			FUN_TcpBufferDataToString(ADR(sReciveMessage),ADR(stReciveData));
			MEMCPY(ADR(sLastStatusCode),ADR(sReciveMessage),2);
			iLastStatusCode := STRING_TO_INT(sLastStatusCode);
			
			IF iLastStatusCode = 1 THEN 
				eCameraGetJobStatus := 1;
				
			ELSIF iLastStatusCode = 0 THEN
				eCameraGetJobStatus := 0;
				
			ELSIF iLastStatusCode = -2 THEN
				eCameraGetJobStatus := -2;
				
			END_IF	
			eCameraMethodState := CAMERA_METHOD_SEND_COMMAND;
			eCameraState := CAMERA_METHOD_DONE;

		END_IF
END_CASE
END_METHOD

METHOD PROTECTED MS_GetOnline
CASE eCameraMethodState OF
	CAMERA_METHOD_SEND_COMMAND:
		MEMSET(ADR(sSendMessage),0,SIZEOF(sSendMessage));
		sSendMessage := 'GO$R$L';
		FUN_StringToTcpBufferData(ADR(sSendMessage),ADR(stSendData));
		
		IF fbTcpClient.MR_AppendToSendBuffer(stSendData) THEN
			eCameraMethodState := CAMERA_METHOD_RECEIVE_RESPONSE;
							
		END_IF

	CAMERA_METHOD_RECEIVE_RESPONSE:
		stReciveData := fbTcpClient.NextRecivedMessage;
		
		IF stReciveData.iLength > 0 THEN
			MEMSET(ADR(sReciveMessage),0,SIZEOF(sReciveMessage));
			FUN_TcpBufferDataToString(ADR(sReciveMessage),ADR(stReciveData));
			MEMCPY(ADR(sLastStatusCode),ADR(sReciveMessage),2);
			iLastStatusCode := STRING_TO_INT(sLastStatusCode);
			
			IF iLastStatusCode = 0 THEN 
				eCameraGetOnlineStatus := 0;
				
			ELSIF iLastStatusCode = 1 THEN
				eCameraGetOnlineStatus := 1;
				
			END_IF	
			eCameraMethodState := CAMERA_METHOD_SEND_COMMAND;
			eCameraState := CAMERA_METHOD_DONE;

		END_IF
END_CASE
END_METHOD

METHOD PROTECTED MS_GetPosition
CASE eCameraGetPositionState OF
	CAMERA_GET_POSITION_SEND_COMMAND_X:
		MEMSET(ADR(sSendMessage),0,SIZEOF(sSendMessage));
		sSendMessage := FUN_MergeStrings3('GV', sPositionXVariable,'$R$L');
		FUN_StringToTcpBufferData(ADR(sSendMessage),ADR(stSendData));
		
		IF fbTcpClient.MR_AppendToSendBuffer(stSendData) THEN
			eCameraGetPositionState := CAMERA_GET_POSITION_RECEIVE_RESPONSE_X;
							
		END_IF

	CAMERA_GET_POSITION_RECEIVE_RESPONSE_X:
		stReciveData := fbTcpClient.NextRecivedMessage;
		
		IF stReciveData.iLength > 0 THEN
			MEMSET(ADR(sReciveMessage),0,SIZEOF(sReciveMessage));
			FUN_TcpBufferDataToString(ADR(sReciveMessage),ADR(stReciveData));
			MEMCPY(ADR(sLastStatusCode),ADR(sReciveMessage),2);
			iLastStatusCode := STRING_TO_INT(sLastStatusCode);
			
			IF iLastStatusCode = 1 THEN 
				eCameraGetPositionStatus := 1;
				sPositionString := TO_STRING(sReciveMessage);
				sPositionStringDel := DELETE(sPositionString,3,1);
				lrPositionX := STRING_TO_LREAL(sPositionStringDel);
				
			ELSIF iLastStatusCode = 0 THEN
				eCameraGetPositionStatus := 0;
				
			ELSIF iLastStatusCode = -1 THEN
				eCameraGetPositionStatus := -1;
				
			ELSIF iLastStatusCode = -2 THEN
				eCameraGetPositionStatus := -2;
				
			END_IF	
			eCameraGetPositionState := CAMERA_GET_POSITION_SEND_COMMAND_Y;

		END_IF
	
	CAMERA_GET_POSITION_SEND_COMMAND_Y:
		MEMSET(ADR(sSendMessage),0,SIZEOF(sSendMessage));
		sSendMessage := FUN_MergeStrings3('GV', sPositionYVariable,'$R$L');
		FUN_StringToTcpBufferData(ADR(sSendMessage),ADR(stSendData));
		
		IF fbTcpClient.MR_AppendToSendBuffer(stSendData) THEN
			eCameraGetPositionState := CAMERA_GET_POSITION_RECEIVE_RESPONSE_Y;
							
		END_IF

	CAMERA_GET_POSITION_RECEIVE_RESPONSE_Y:
		stReciveData := fbTcpClient.NextRecivedMessage;
		
		IF stReciveData.iLength > 0 THEN
			MEMSET(ADR(sReciveMessage),0,SIZEOF(sReciveMessage));
			FUN_TcpBufferDataToString(ADR(sReciveMessage),ADR(stReciveData));
			MEMCPY(ADR(sLastStatusCode),ADR(sReciveMessage),2);
			iLastStatusCode := STRING_TO_INT(sLastStatusCode);
			
			IF iLastStatusCode = 1 THEN 
				eCameraGetPositionStatus := 1;
				sPositionString := TO_STRING(sReciveMessage);
				sPositionStringDel := DELETE(sPositionString,3,1);
				lrPositionY := STRING_TO_LREAL(sPositionStringDel);
				
			ELSIF iLastStatusCode = 0 THEN
				eCameraGetPositionStatus := 0;
				
			ELSIF iLastStatusCode = -1 THEN
				eCameraGetPositionStatus := -1;
				
			ELSIF iLastStatusCode = -2 THEN
				eCameraGetPositionStatus := -2;
				
			END_IF	
			eCameraGetPositionState := CAMERA_GET_POSITION_SEND_COMMAND_ROTATION;
			
		END_IF
		
		
	CAMERA_GET_POSITION_SEND_COMMAND_ROTATION:
		MEMSET(ADR(sSendMessage),0,SIZEOF(sSendMessage));
		sSendMessage := FUN_MergeStrings3('GV', sRotationVariable,'$R$L');
		FUN_StringToTcpBufferData(ADR(sSendMessage),ADR(stSendData));
		
		IF fbTcpClient.MR_AppendToSendBuffer(stSendData) THEN
			eCameraGetPositionState := CAMERA_GET_POSITION_RECEIVE_RESPONSE_ROTATION;
							
		END_IF

	CAMERA_GET_POSITION_RECEIVE_RESPONSE_ROTATION:
		stReciveData := fbTcpClient.NextRecivedMessage;
		
		IF stReciveData.iLength > 0 THEN
			MEMSET(ADR(sReciveMessage),0,SIZEOF(sReciveMessage));
			FUN_TcpBufferDataToString(ADR(sReciveMessage),ADR(stReciveData));
			MEMCPY(ADR(sLastStatusCode),ADR(sReciveMessage),2);
			iLastStatusCode := STRING_TO_INT(sLastStatusCode);
			
			IF iLastStatusCode = 1 THEN 
				eCameraGetPositionStatus := 1;
				sPositionString := TO_STRING(sReciveMessage);
				sPositionStringDel := DELETE(sPositionString,3,1);
				lrRotation := STRING_TO_LREAL(sPositionStringDel);
				
			ELSIF iLastStatusCode = 0 THEN
				eCameraGetPositionStatus := 0;
				
			ELSIF iLastStatusCode = -1 THEN
				eCameraGetPositionStatus := -1;
				
			ELSIF iLastStatusCode = -2 THEN
				eCameraGetPositionStatus := -2;
				
			END_IF	
			eCameraGetPositionState := CAMERA_GET_POSITION_GETTING_DONE;

		END_IF
		
	CAMERA_GET_POSITION_GETTING_DONE:
		IF lrPositionX = 0.0 AND lrPositionY = 0.0 THEN
			eCameraGetPositionStatus := -3;
			
		END_IF
		eCameraGetPositionState := CAMERA_GET_POSITION_SEND_COMMAND_X;
		eCameraState := CAMERA_METHOD_DONE;
		
END_CASE
END_METHOD

METHOD PROTECTED MS_GetValueEasyBuilder
CASE eCameraMethodState OF
	CAMERA_METHOD_SEND_COMMAND:
		MEMSET(ADR(sSendMessage),0,SIZEOF(sSendMessage));
		sSendMessage := FUN_MergeStrings3('GV', sEasyBuilderValueName,'$R$L');
		FUN_StringToTcpBufferData(ADR(sSendMessage),ADR(stSendData));
		
		IF fbTcpClient.MR_AppendToSendBuffer(stSendData) THEN
			eCameraMethodState := CAMERA_METHOD_RECEIVE_RESPONSE;
							
		END_IF

	CAMERA_METHOD_RECEIVE_RESPONSE:
		stReciveData := fbTcpClient.NextRecivedMessage;
		
		IF stReciveData.iLength > 0 THEN
			MEMSET(ADR(sReciveMessage),0,SIZEOF(sReciveMessage));
			FUN_TcpBufferDataToString(ADR(sReciveMessage),ADR(stReciveData));
			MEMCPY(ADR(sLastStatusCode),ADR(sReciveMessage),2);
			iLastStatusCode := STRING_TO_INT(sLastStatusCode);
			
			IF iLastStatusCode = 1 THEN 
				eCameraGetValueEasyBuilderStatus := 1;
				
			ELSIF iLastStatusCode = 0 THEN
				eCameraGetValueEasyBuilderStatus := 0;
				
			ELSIF iLastStatusCode = -1 THEN
				eCameraGetValueEasyBuilderStatus := -1;
				
			ELSIF iLastStatusCode = -2 THEN
				eCameraGetValueEasyBuilderStatus := -2;
				
			END_IF	
			eCameraMethodState := CAMERA_METHOD_SEND_COMMAND;
			eCameraState := CAMERA_METHOD_DONE;

		END_IF
END_CASE
END_METHOD

METHOD PROTECTED MS_GetValues
CASE eCameraGetValuesState OF
	CAMERA_GET_VALUES_SEND_COMMAND_VALUE_1:
		MEMSET(ADR(sSendMessage),0,SIZEOF(sSendMessage));
		sSendMessage := FUN_MergeStrings3('GV', sVariable1,'$R$L');
		FUN_StringToTcpBufferData(ADR(sSendMessage),ADR(stSendData));
		
		IF fbTcpClient.MR_AppendToSendBuffer(stSendData) THEN
			eCameraGetValuesState := CAMERA_GET_VALUES_RECEIVE_RESPONSE_VALUE_1;
							
		END_IF

	CAMERA_GET_VALUES_RECEIVE_RESPONSE_VALUE_1:
		stReciveData := fbTcpClient.NextRecivedMessage;
		
		IF stReciveData.iLength > 0 THEN
			MEMSET(ADR(sReciveMessage),0,SIZEOF(sReciveMessage));
			FUN_TcpBufferDataToString(ADR(sReciveMessage),ADR(stReciveData));
			MEMCPY(ADR(sLastStatusCode),ADR(sReciveMessage),2);
			iLastStatusCode := STRING_TO_INT(sLastStatusCode);
			
			IF iLastStatusCode = 1 THEN 
				eCameraGetValuesStatus := 1;
				sPositionString := TO_STRING(sReciveMessage);
				sPositionStringDel := DELETE(sPositionString,3,1);
				lrValue1 := STRING_TO_LREAL(sPositionStringDel);
				
			ELSIF iLastStatusCode = 0 THEN
				eCameraGetValuesStatus := 0;
				
			ELSIF iLastStatusCode = -1 THEN
				eCameraGetValuesStatus := -1;
				
			ELSIF iLastStatusCode = -2 THEN
				eCameraGetValuesStatus := -2;
				
			END_IF	
			eCameraGetValuesState := CAMERA_GET_VALUES_SEND_COMMAND_VALUE_2;

		END_IF
	
	CAMERA_GET_VALUES_SEND_COMMAND_VALUE_2:
		MEMSET(ADR(sSendMessage),0,SIZEOF(sSendMessage));
		sSendMessage := FUN_MergeStrings3('GV', sVariable2,'$R$L');
		FUN_StringToTcpBufferData(ADR(sSendMessage),ADR(stSendData));
		
		IF fbTcpClient.MR_AppendToSendBuffer(stSendData) THEN
			eCameraGetValuesState := CAMERA_GET_VALUES_RECEIVE_RESPONSE_VALUE_2;
							
		END_IF

	CAMERA_GET_VALUES_RECEIVE_RESPONSE_VALUE_2:
		stReciveData := fbTcpClient.NextRecivedMessage;
		
		IF stReciveData.iLength > 0 THEN
			MEMSET(ADR(sReciveMessage),0,SIZEOF(sReciveMessage));
			FUN_TcpBufferDataToString(ADR(sReciveMessage),ADR(stReciveData));
			MEMCPY(ADR(sLastStatusCode),ADR(sReciveMessage),2);
			iLastStatusCode := STRING_TO_INT(sLastStatusCode);
			
			IF iLastStatusCode = 1 THEN 
				eCameraGetValuesStatus := 1;
				sPositionString := TO_STRING(sReciveMessage);
				sPositionStringDel := DELETE(sPositionString,3,1);
				lrValue2 := STRING_TO_LREAL(sPositionStringDel);
				
			ELSIF iLastStatusCode = 0 THEN
				eCameraGetValuesStatus := 0;
				
			ELSIF iLastStatusCode = -1 THEN
				eCameraGetValuesStatus := -1;
				
			ELSIF iLastStatusCode = -2 THEN
				eCameraGetValuesStatus := -2;
				
			END_IF	
			eCameraGetValuesState := CAMERA_GET_VALUES_SEND_COMMAND_VALUE_3;
			
		END_IF
		
		
	CAMERA_GET_VALUES_SEND_COMMAND_VALUE_3:
		MEMSET(ADR(sSendMessage),0,SIZEOF(sSendMessage));
		sSendMessage := FUN_MergeStrings3('GV', sVariable3,'$R$L');
		FUN_StringToTcpBufferData(ADR(sSendMessage),ADR(stSendData));
		
		IF fbTcpClient.MR_AppendToSendBuffer(stSendData) THEN
			eCameraGetValuesState := CAMERA_GET_VALUES_RECEIVE_RESPONSE_VALUE_3;

		END_IF

	CAMERA_GET_VALUES_RECEIVE_RESPONSE_VALUE_3:
		stReciveData := fbTcpClient.NextRecivedMessage;
		
		IF stReciveData.iLength > 0 THEN
			MEMSET(ADR(sReciveMessage),0,SIZEOF(sReciveMessage));
			FUN_TcpBufferDataToString(ADR(sReciveMessage),ADR(stReciveData));
			MEMCPY(ADR(sLastStatusCode),ADR(sReciveMessage),2);
			iLastStatusCode := STRING_TO_INT(sLastStatusCode);
			
			IF iLastStatusCode = 1 THEN 
				eCameraGetValuesStatus := 1;
				sPositionString := TO_STRING(sReciveMessage);
				sPositionStringDel := DELETE(sPositionString,3,1);
				lrValue3 := STRING_TO_LREAL(sPositionStringDel);
				
			ELSIF iLastStatusCode = 0 THEN
				eCameraGetValuesStatus := 0;
				
			ELSIF iLastStatusCode = -1 THEN
				eCameraGetValuesStatus := -1;
				
			ELSIF iLastStatusCode = -2 THEN
				eCameraGetValuesStatus := -2;
				
			END_IF	
			eCameraGetValuesState := CAMERA_GET_VALUES_SEND_COMMAND_VALUE_4;

		END_IF


	CAMERA_GET_VALUES_SEND_COMMAND_VALUE_4:
		MEMSET(ADR(sSendMessage),0,SIZEOF(sSendMessage));
		sSendMessage := FUN_MergeStrings3('GV', sVariable4,'$R$L');
		FUN_StringToTcpBufferData(ADR(sSendMessage),ADR(stSendData));
		
		IF fbTcpClient.MR_AppendToSendBuffer(stSendData) THEN
			eCameraGetValuesState := CAMERA_GET_VALUES_RECEIVE_RESPONSE_VALUE_4;
							
		END_IF

	CAMERA_GET_VALUES_RECEIVE_RESPONSE_VALUE_4:
		stReciveData := fbTcpClient.NextRecivedMessage;
		
		IF stReciveData.iLength > 0 THEN
			MEMSET(ADR(sReciveMessage),0,SIZEOF(sReciveMessage));
			FUN_TcpBufferDataToString(ADR(sReciveMessage),ADR(stReciveData));
			MEMCPY(ADR(sLastStatusCode),ADR(sReciveMessage),2);
			iLastStatusCode := STRING_TO_INT(sLastStatusCode);
			
			IF iLastStatusCode = 1 THEN 
				eCameraGetValuesStatus := 1;
				sPositionString := TO_STRING(sReciveMessage);
				sPositionStringDel := DELETE(sPositionString,3,1);
				lrValue4 := STRING_TO_LREAL(sPositionStringDel);
				
			ELSIF iLastStatusCode = 0 THEN
				eCameraGetValuesStatus := 0;
				
			ELSIF iLastStatusCode = -1 THEN
				eCameraGetValuesStatus := -1;
				
			ELSIF iLastStatusCode = -2 THEN
				eCameraGetValuesStatus := -2;
				
			END_IF	
			eCameraGetValuesState := CAMERA_GET_VALUES_GETTING_DONE;

		END_IF
		
	CAMERA_GET_VALUES_GETTING_DONE:
		
		IF lrValue1 = 0.0 OR lrValue2 = 0.0 OR lrValue3 = 0.0 OR lrValue4 = 0.0 THEN
			eCameraGetValuesStatus := -3;
			
		END_IF
		eCameraGetValuesState := CAMERA_GET_VALUES_SEND_COMMAND_VALUE_1;
		eCameraState := CAMERA_METHOD_DONE;
		
END_CASE
END_METHOD

METHOD PROTECTED MS_GetValueSpreadsheet
CASE eCameraMethodState OF
	CAMERA_METHOD_SEND_COMMAND:
		MEMSET(ADR(sSendMessage),0,SIZEOF(sSendMessage));
		sSendMessage := FUN_MergeStrings5('GV', TO_STRING(iColumnValueSpreadsheet), TO_STRING(iRowValueSpreadsheet), '$R$L', '');
		FUN_StringToTcpBufferData(ADR(sSendMessage),ADR(stSendData));
		
		IF fbTcpClient.MR_AppendToSendBuffer(stSendData) THEN
			eCameraMethodState := CAMERA_METHOD_RECEIVE_RESPONSE;
							
		END_IF

	CAMERA_METHOD_RECEIVE_RESPONSE:
		stReciveData := fbTcpClient.NextRecivedMessage;
		
		IF stReciveData.iLength > 0 THEN
			MEMSET(ADR(sReciveMessage),0,SIZEOF(sReciveMessage));
			FUN_TcpBufferDataToString(ADR(sReciveMessage),ADR(stReciveData));
			MEMCPY(ADR(sLastStatusCode),ADR(sReciveMessage),2);
			iLastStatusCode := STRING_TO_INT(sLastStatusCode);
			
			IF iLastStatusCode = 1 THEN 
				eCameraGetValueSpreadsheetStatus := 1;
				
			ELSIF iLastStatusCode = 0 THEN
				eCameraGetValueSpreadsheetStatus := 0;
				
			ELSIF iLastStatusCode = -1 THEN
				eCameraGetValueSpreadsheetStatus := -1;
				
			ELSIF iLastStatusCode = -2 THEN
				eCameraGetValueSpreadsheetStatus := -2;
				
			END_IF	
			eCameraMethodState := CAMERA_METHOD_SEND_COMMAND;
			eCameraState := CAMERA_METHOD_DONE;

		END_IF
END_CASE
END_METHOD

METHOD PROTECTED MS_Idle
;
END_METHOD

METHOD PROTECTED MS_ImageTrigger
CASE eCameraMethodState OF
	CAMERA_METHOD_SEND_COMMAND:
		MEMSET(ADR(sSendMessage),0,SIZEOF(sSendMessage));
		sSendMessage := 'SW8$R$L';
		FUN_StringToTcpBufferData(ADR(sSendMessage),ADR(stSendData));
		
		IF fbTcpClient.MR_AppendToSendBuffer(stSendData) THEN
			eCameraMethodState := CAMERA_METHOD_RECEIVE_RESPONSE;
							
		END_IF

	CAMERA_METHOD_RECEIVE_RESPONSE:
		stReciveData := fbTcpClient.NextRecivedMessage;
		
		IF stReciveData.iLength > 0 THEN
			MEMSET(ADR(sReciveMessage),0,SIZEOF(sReciveMessage));
			FUN_TcpBufferDataToString(ADR(sReciveMessage),ADR(stReciveData));
			MEMCPY(ADR(sLastStatusCode),ADR(sReciveMessage),2);
			iLastStatusCode := STRING_TO_INT(sLastStatusCode);
			
			IF iLastStatusCode = 1 THEN 
				eCameraImageTriggerStatus := 1;
				
			ELSIF iLastStatusCode = 0 THEN
				eCameraImageTriggerStatus := 0;
				
			ELSIF iLastStatusCode = -1 THEN
				eCameraImageTriggerStatus := -1;
				
			ELSIF iLastStatusCode = -2 THEN
				eCameraImageTriggerStatus := -2;
				
			ELSIF iLastStatusCode = -6 THEN
				eCameraImageTriggerStatus := -6;
				
			END_IF	
			eCameraMethodState := CAMERA_METHOD_SEND_COMMAND;			
			eCameraState := CAMERA_METHOD_DONE;

		END_IF
END_CASE
END_METHOD

METHOD PROTECTED MS_Initializing //C:\TwinCAT\log\filelog.txt
VAR_INST
//	tClearBuffers		:	TON;
END_VAR
CASE eCameraInitState OF
	CAMERA_INIT_CONNECTION:
		fbTcpClient.MR_Init();
		
		IF fbTcpClient.Active THEN
			eCameraInitState := CAMERA_INIT_CLEAR_BUFFER;	
			
		ELSIF fbTcpClient.Error THEN
			bError := TRUE;
			iErrorID := fbTcpClient.ErrorID;
			
		END_IF
		
	CAMERA_INIT_CLEAR_BUFFER:
		fbTcpClient.MR_ClearAllBuffers();
		eCameraInitState := CAMERA_INIT_WAIT_FOR_USERNAME;
		
		IF fbTcpClient.Error THEN
			bError := TRUE;
			iErrorID := fbTcpClient.ErrorID;
			
		END_IF
		
	CAMERA_INIT_WAIT_FOR_USERNAME: 
		stReciveData := fbTcpClient.NextRecivedMessage;
		
		IF stReciveData.iLength > 0 THEN
			MEMSET(ADR(sReciveMessage),0,SIZEOF(sReciveMessage));
			FUN_TcpBufferDataToString(ADR(sReciveMessage),ADR(stReciveData));		
	
			IF RIGHT(sReciveMessage, 6) = 'User: ' THEN	
				eCameraInitState := CAMERA_INIT_WRITE_USER;
			
			END_IF
		ELSIF fbTcpClient.Error THEN
			bError := TRUE;
			iErrorID := fbTcpClient.ErrorID;
			
		END_IF
			
	CAMERA_INIT_WRITE_USER:
		MEMSET(ADR(sSendMessage),0,SIZEOF(sSendMessage));
		sSendMessage := 'admin$R$L';
		FUN_StringToTcpBufferData(ADR(sSendMessage),ADR(stSendData));
		stSendData.iLength := INT_TO_UDINT(LEN(sSendMessage));
		
		IF fbTcpClient.MR_AppendToSendBuffer(stSendData) THEN
			eCameraInitState := CAMERA_INIT_WAIT_FOR_PASSWORD;
		
		ELSIF fbTcpClient.Error THEN
			bError := TRUE;
			iErrorID := fbTcpClient.ErrorID;
			
		END_IF
		
	CAMERA_INIT_WAIT_FOR_PASSWORD:
		stReciveData := fbTcpClient.NextRecivedMessage;
		
		IF stReciveData.iLength > 0 THEN
			MEMSET(ADR(sReciveMessage),0,SIZEOF(sReciveMessage));
			FUN_TcpBufferDataToString(ADR(sReciveMessage),ADR(stReciveData));
			
			IF sReciveMessage = 'Password: ' THEN		
				eCameraInitState := CAMERA_INIT_WRITE_PASSWORD;
			
			END_IF
		ELSIF fbTcpClient.Error THEN
			bError := TRUE;
			iErrorID := fbTcpClient.ErrorID;
			
		END_IF

	CAMERA_INIT_WRITE_PASSWORD:
		MEMSET(ADR(sSendMessage),0,SIZEOF(sSendMessage));
		sSendMessage := '$R$L';
		FUN_StringToTcpBufferData(ADR(sSendMessage),ADR(stSendData));
		stSendData.iLength := INT_TO_UDINT(LEN(sSendMessage));
		
		IF fbTcpClient.MR_AppendToSendBuffer(stSendData) THEN
			eCameraInitState := CAMERA_INIT_WAIT_FOR_CONFIRMATION;

		ELSIF fbTcpClient.Error THEN
			bError := TRUE;
			iErrorID := fbTcpClient.ErrorID;
			
		END_IF
		
	CAMERA_INIT_WAIT_FOR_CONFIRMATION:
		stReciveData := fbTcpClient.NextRecivedMessage;
		
		IF stReciveData.iLength > 0 THEN
			MEMSET(ADR(sReciveMessage),0,SIZEOF(sReciveMessage));
			FUN_TcpBufferDataToString(ADR(sReciveMessage),ADR(stReciveData));
	
			IF sReciveMessage = 'User Logged In$R$L' THEN		
				eCameraInitState := CAMERA_INIT_DONE;
			
			END_IF
		ELSIF fbTcpClient.Error THEN
			bError := TRUE;
			iErrorID := fbTcpClient.ErrorID;
			
		END_IF
		
	CAMERA_INIT_DONE:
		eCameraInitState := CAMERA_INIT_CONNECTION;
		eCameraState := CAMERA_READY;
			
END_CASE
END_METHOD

METHOD PROTECTED MS_LoadFile
CASE eCameraMethodState OF
	CAMERA_METHOD_SEND_COMMAND:
		MEMSET(ADR(sSendMessage),0,SIZEOF(sSendMessage));
		sSendMessage := FUN_MergeStrings3('LF', sLoadFileName,'$R$L');
		FUN_StringToTcpBufferData(ADR(sSendMessage),ADR(stSendData));
		
		IF fbTcpClient.MR_AppendToSendBuffer(stSendData) THEN
			eCameraMethodState := CAMERA_METHOD_RECEIVE_RESPONSE;
							
		END_IF

	CAMERA_METHOD_RECEIVE_RESPONSE:
		stReciveData := fbTcpClient.NextRecivedMessage;
		
		IF stReciveData.iLength > 0 THEN
			MEMSET(ADR(sReciveMessage),0,SIZEOF(sReciveMessage));
			FUN_TcpBufferDataToString(ADR(sReciveMessage),ADR(stReciveData));
			MEMCPY(ADR(sLastStatusCode),ADR(sReciveMessage),2);
			iLastStatusCode := STRING_TO_INT(sLastStatusCode);
			
			IF iLastStatusCode = 1 THEN 
				eCameraLoadFileStatus := 1;
				
			ELSIF iLastStatusCode = 0 THEN
				eCameraLoadFileStatus := 0;
				
			ELSIF iLastStatusCode = -1 THEN
				eCameraLoadFileStatus := -1;
				
			ELSIF iLastStatusCode = -2 THEN
				eCameraLoadFileStatus := -2;
				
			ELSIF iLastStatusCode = -4 THEN
				eCameraLoadFileStatus := -4;
				
			ELSIF iLastStatusCode = -6 THEN
				eCameraLoadFileStatus := -6;
				
			END_IF	
			eCameraMethodState := CAMERA_METHOD_SEND_COMMAND;
			eCameraState := CAMERA_METHOD_DONE;

		END_IF
END_CASE
END_METHOD

METHOD PROTECTED MS_MethodDone
VAR_INPUT
END_VAR
IF NOT bBusy THEN
	eCameraState := CAMERA_IDLE;
	
END_IF
END_METHOD

METHOD PROTECTED MS_PutLive
CASE eCameraMethodState OF
	CAMERA_METHOD_SEND_COMMAND:
		MEMSET(ADR(sSendMessage),0,SIZEOF(sSendMessage));
		sSendMessage := FUN_MergeStrings3('Put live ', TO_STRING(bEnableLiveAcquisition), '$R$L');
		FUN_StringToTcpBufferData(ADR(sSendMessage),ADR(stSendData));
		
		IF fbTcpClient.MR_AppendToSendBuffer(stSendData) THEN
			eCameraMethodState := CAMERA_METHOD_RECEIVE_RESPONSE;
							
		END_IF

	CAMERA_METHOD_RECEIVE_RESPONSE:
		stReciveData := fbTcpClient.NextRecivedMessage;
		
		IF stReciveData.iLength > 0 THEN
			MEMSET(ADR(sReciveMessage),0,SIZEOF(sReciveMessage));
			FUN_TcpBufferDataToString(ADR(sReciveMessage),ADR(stReciveData));
			MEMCPY(ADR(sLastStatusCode),ADR(sReciveMessage),2);
			iLastStatusCode := STRING_TO_INT(sLastStatusCode);
			
			IF iLastStatusCode = 1 THEN 
				eCameraPutLiveStatus := 1;
				
			ELSIF iLastStatusCode = 0 THEN
				eCameraPutLiveStatus := 0;
				
			ELSIF iLastStatusCode = -1 THEN
				eCameraPutLiveStatus := -1;
				
			ELSIF iLastStatusCode = -2 THEN
				eCameraPutLiveStatus := -2;
				
			ELSIF iLastStatusCode = -6 THEN
				eCameraPutLiveStatus := -6;
				
			END_IF	
			eCameraMethodState := CAMERA_METHOD_SEND_COMMAND;
			eCameraState := CAMERA_METHOD_DONE;

		END_IF
END_CASE
END_METHOD

METHOD PROTECTED MS_PutPortnum
CASE eCameraMethodState OF
	CAMERA_METHOD_SEND_COMMAND:
		MEMSET(ADR(sSendMessage),0,SIZEOF(sSendMessage));
		sSendMessage := FUN_MergeStrings3('Put Portnum ', TO_STRING(iPortNumber), '$R$L');
		FUN_StringToTcpBufferData(ADR(sSendMessage),ADR(stSendData));
		
		IF fbTcpClient.MR_AppendToSendBuffer(stSendData) THEN
			eCameraMethodState := CAMERA_METHOD_RECEIVE_RESPONSE;
							
		END_IF

	CAMERA_METHOD_RECEIVE_RESPONSE:
		stReciveData := fbTcpClient.NextRecivedMessage;
		
		IF stReciveData.iLength > 0 THEN
			MEMSET(ADR(sReciveMessage),0,SIZEOF(sReciveMessage));
			FUN_TcpBufferDataToString(ADR(sReciveMessage),ADR(stReciveData));
			MEMCPY(ADR(sLastStatusCode),ADR(sReciveMessage),2);
			iLastStatusCode := STRING_TO_INT(sLastStatusCode);
			
			IF iLastStatusCode = 1 THEN 
				eCameraPutPortnumStatus := 1;
				
			ELSIF iLastStatusCode = 0 THEN
				eCameraPutPortnumStatus := 0;
				
			ELSIF iLastStatusCode = -1 THEN
				eCameraPutPortnumStatus := -1;
				
			ELSIF iLastStatusCode = -2 THEN
				eCameraPutPortnumStatus := -2;
				
			ELSIF iLastStatusCode = -6 THEN
				eCameraPutPortnumStatus := -6;
				
			END_IF	
			eCameraMethodState := CAMERA_METHOD_SEND_COMMAND;
			eCameraState := CAMERA_METHOD_DONE;

		END_IF
END_CASE
END_METHOD

METHOD PROTECTED MS_PutTimeout
CASE eCameraMethodState OF
	CAMERA_METHOD_SEND_COMMAND:
		MEMSET(ADR(sSendMessage),0,SIZEOF(sSendMessage));
		sSendMessage := FUN_MergeStrings3('Put Timeout ', TO_STRING(iTimeout), '$R$L');
		FUN_StringToTcpBufferData(ADR(sSendMessage),ADR(stSendData));
		
		IF fbTcpClient.MR_AppendToSendBuffer(stSendData) THEN
			eCameraMethodState := CAMERA_METHOD_RECEIVE_RESPONSE;
							
		END_IF

	CAMERA_METHOD_RECEIVE_RESPONSE:
		stReciveData := fbTcpClient.NextRecivedMessage;
		
		IF stReciveData.iLength > 0 THEN
			MEMSET(ADR(sReciveMessage),0,SIZEOF(sReciveMessage));
			FUN_TcpBufferDataToString(ADR(sReciveMessage),ADR(stReciveData));
			MEMCPY(ADR(sLastStatusCode),ADR(sReciveMessage),2);
			iLastStatusCode := STRING_TO_INT(sLastStatusCode);
			
			IF iLastStatusCode = 1 THEN 
				eCameraPutTimeoutStatus := 1;
				
			ELSIF iLastStatusCode = 0 THEN
				eCameraPutTimeoutStatus := 0;
				
			ELSIF iLastStatusCode = -1 THEN
				eCameraPutTimeoutStatus := -1;
				
			ELSIF iLastStatusCode = -6 THEN
				eCameraPutTimeoutStatus := -6;
				
			END_IF	
			eCameraMethodState := CAMERA_METHOD_SEND_COMMAND;
			eCameraState := CAMERA_METHOD_DONE;
			
		END_IF
END_CASE
END_METHOD

METHOD PROTECTED MS_PutUpdate
CASE eCameraMethodState OF
	CAMERA_METHOD_SEND_COMMAND:
		MEMSET(ADR(sSendMessage),0,SIZEOF(sSendMessage));
		sSendMessage := FUN_MergeStrings3('Put Update ', TO_STRING(iUpdateNumber), '$R$L');
		FUN_StringToTcpBufferData(ADR(sSendMessage),ADR(stSendData));
		
		IF fbTcpClient.MR_AppendToSendBuffer(stSendData) THEN
			eCameraMethodState := CAMERA_METHOD_RECEIVE_RESPONSE;
							
		END_IF

	CAMERA_METHOD_RECEIVE_RESPONSE:
		stReciveData := fbTcpClient.NextRecivedMessage;
		
		IF stReciveData.iLength > 0 THEN
			MEMSET(ADR(sReciveMessage),0,SIZEOF(sReciveMessage));
			FUN_TcpBufferDataToString(ADR(sReciveMessage),ADR(stReciveData));
			MEMCPY(ADR(sLastStatusCode),ADR(sReciveMessage),2);
			iLastStatusCode := STRING_TO_INT(sLastStatusCode);
			
			IF iLastStatusCode = 1 THEN 
				eCameraPutUpdateStatus := 1;
				
			ELSIF iLastStatusCode = 0 THEN
				eCameraPutUpdateStatus := 0;
				
			ELSIF iLastStatusCode = -1 THEN
				eCameraPutUpdateStatus := -1;
				
			ELSIF iLastStatusCode = -2 THEN
				eCameraPutUpdateStatus := -2;
				
			ELSIF iLastStatusCode = -6 THEN
				eCameraPutUpdateStatus := -6;
				
			END_IF	
			eCameraMethodState := CAMERA_METHOD_SEND_COMMAND;
			eCameraState := CAMERA_METHOD_DONE;

		END_IF
END_CASE
END_METHOD

METHOD PROTECTED MS_PutWatch
CASE eCameraMethodState OF
	CAMERA_METHOD_SEND_COMMAND:
		MEMSET(ADR(sSendMessage),0,SIZEOF(sSendMessage));
		sSendMessage := FUN_MergeStrings5('Put Watch ', TO_STRING(iColumnPut), TO_STRING(iRowPut), TO_STRING(iOutputEnable), '$R$L');
		FUN_StringToTcpBufferData(ADR(sSendMessage),ADR(stSendData));
		
		IF fbTcpClient.MR_AppendToSendBuffer(stSendData) THEN
			eCameraMethodState := CAMERA_METHOD_RECEIVE_RESPONSE;
							
		END_IF

	CAMERA_METHOD_RECEIVE_RESPONSE:
		stReciveData := fbTcpClient.NextRecivedMessage;
		
		IF stReciveData.iLength > 0 THEN
			MEMSET(ADR(sReciveMessage),0,SIZEOF(sReciveMessage));
			FUN_TcpBufferDataToString(ADR(sReciveMessage),ADR(stReciveData));
			MEMCPY(ADR(sLastStatusCode),ADR(sReciveMessage),2);
			iLastStatusCode := STRING_TO_INT(sLastStatusCode);
			
			IF iLastStatusCode = 1 THEN 
				eCameraPutWatchStatus := 1;
				
			ELSIF iLastStatusCode = 0 THEN
				eCameraPutWatchStatus := 0;
				
			ELSIF iLastStatusCode = -1 THEN
				eCameraPutWatchStatus := -1;
				
			ELSIF iLastStatusCode = -2 THEN
				eCameraPutWatchStatus := -2;
				
			ELSIF iLastStatusCode = -6 THEN
				eCameraPutWatchStatus := -6;
				
			END_IF	
			eCameraMethodState := CAMERA_METHOD_SEND_COMMAND;
			eCameraState := CAMERA_METHOD_DONE;

		END_IF
END_CASE
END_METHOD

METHOD PROTECTED MS_Ready
VAR_INPUT
END_VAR
eCameraState := CAMERA_IDLE;
END_METHOD

METHOD PROTECTED MS_Reset
VAR_INPUT
END_VAR
IF M_ResetParameters() THEN
	eCameraState := CAMERA_METHOD_DONE;
	
END_IF
END_METHOD

METHOD PROTECTED MS_ResetSystem
CASE eCameraMethodState OF
	CAMERA_METHOD_SEND_COMMAND:
		MEMSET(ADR(sSendMessage),0,SIZEOF(sSendMessage));
		sSendMessage := 'RT$R$L';
		FUN_StringToTcpBufferData(ADR(sSendMessage),ADR(stSendData));
		
		IF fbTcpClient.MR_AppendToSendBuffer(stSendData) THEN
			eCameraMethodState := CAMERA_METHOD_RECEIVE_RESPONSE;
							
		END_IF

	CAMERA_METHOD_RECEIVE_RESPONSE:
		stReciveData := fbTcpClient.NextRecivedMessage;
		
		IF stReciveData.iLength > 0 THEN
			MEMSET(ADR(sReciveMessage),0,SIZEOF(sReciveMessage));
			FUN_TcpBufferDataToString(ADR(sReciveMessage),ADR(stReciveData));
			MEMCPY(ADR(sLastStatusCode),ADR(sReciveMessage),2);
			iLastStatusCode := STRING_TO_INT(sLastStatusCode);
			
			IF iLastStatusCode = -6 THEN 
				eCameraResetSystemStatus := -6;
				
			END_IF	
		ELSE
			eCameraResetSystemStatus := -1;
			
		END_IF
		eCameraMethodState := CAMERA_METHOD_SEND_COMMAND;
		eCameraState := CAMERA_METHOD_DONE;
		
END_CASE
END_METHOD

METHOD PROTECTED MS_SetJob
CASE eCameraMethodState OF
	CAMERA_METHOD_SEND_COMMAND:
		MEMSET(ADR(sSendMessage),0,SIZEOF(sSendMessage));
		sSendMessage := FUN_MergeStrings3('SJ', TO_STRING(iJobNumber), '$R$L');
		FUN_StringToTcpBufferData(ADR(sSendMessage),ADR(stSendData));
		
		IF fbTcpClient.MR_AppendToSendBuffer(stSendData) THEN
			eCameraMethodState := CAMERA_METHOD_RECEIVE_RESPONSE;
							
		END_IF

	CAMERA_METHOD_RECEIVE_RESPONSE:
		stReciveData := fbTcpClient.NextRecivedMessage;
		
		IF stReciveData.iLength > 0 THEN
			MEMSET(ADR(sReciveMessage),0,SIZEOF(sReciveMessage));
			FUN_TcpBufferDataToString(ADR(sReciveMessage),ADR(stReciveData));
			MEMCPY(ADR(sLastStatusCode),ADR(sReciveMessage),2);
			iLastStatusCode := STRING_TO_INT(sLastStatusCode);
			
			IF iLastStatusCode = 1 THEN 
				eCameraSetJobStatus := 1;
				
			ELSIF iLastStatusCode = 0 THEN
				eCameraSetJobStatus := 0;
				
			ELSIF iLastStatusCode = -1 THEN
				eCameraSetJobStatus := -1;
				
			ELSIF iLastStatusCode = -2 THEN
				eCameraSetJobStatus := -2;
				
			ELSIF iLastStatusCode = -4 THEN
				eCameraSetJobStatus := -4;
				
			ELSIF iLastStatusCode = -6 THEN
				eCameraSetJobStatus := -6;
				
